PGM546_DRIFT 546.00 BOOL  ; PAST23 TIL T2009
PGM546_DRIFT_N5 2831.09 BOOL
PGM546_FEIL 546.04 BOOL  ; PAST23 TIL T2009
PGM546_FEILTID 546.05 BOOL  ; PAST23 TIL T2009
PGM546_FEILTID_S T0546 BOOL
PGM546_FEILTID_T 0546 NUMBER
PGM546_IKKE_FEIL_N5 2831.13 BOOL
PGM546_START 546.07 BOOL  ; PAST23 TIL T2009
PGM546_STOPP 546.09 BOOL  ; PAST23 TIL T2009
PGM546_STOPP_N5 2831.08 BOOL
PGM546_T2009_DREN_IND 1246.01 BOOL  ; DREN FRA V2347
PGM546_T2009_IND 1246.00 BOOL
PGM548_0_STATUS 548.01 BOOL  ; LAGER TIL T2030-DIREKTE-CONTAINER
PGM548_1_STATUS 548.02 BOOL  ; LAGER TIL T2030-DIREKTE-CONTAINER
PGM548_2030_IND 1248.00 BOOL
PGM548_2_STATUS 548.03 BOOL  ; LAGER TIL T2030-DIREKTE-CONTAINER
PGM548_CONT_IND 1248.02 BOOL
PGM548_DRIFT 548.00 BOOL  ; LAGER TIL T2030-DIREKTE-CONTAINER
PGM548_FEIL 548.04 BOOL  ; LAGER TIL T2030-DIREKTE-CONTAINER
PGM548_FEILTID 548.05 BOOL  ; LAGER TIL T2030-DIREKTE-CONTAINER
PGM548_INDIVID_INNE 548.15 BOOL  ; LAGER TIL T2030-DIREKTE-CONTAINER
PGM548_INDKON 548.06 BOOL  ; LAGER TIL T2030-DIREKTE-CONTAINER
PGM548_MODN_IND 1248.01 BOOL
PGM548_OFF_IMP 548.14 BOOL  ; LAGER TIL T2030-DIREKTE-CONTAINER
PGM548_ONIMPULS 548.11 BOOL  ; LAGER TIL T2030-DIREKTE-CONTAINER
PGM548_START 548.07 BOOL  ; LAGER TIL T2030-DIREKTE-CONTAINER
PGM548_STARTIMPULS 548.10 BOOL  ; LAGER TIL T2030-DIREKTE-CONTAINER
PGM548_STOPP 548.09 BOOL  ; LAGER TIL T2030-DIREKTE-CONTAINER
PGM548_TID_S T0548 BOOL  ; X
PGM548_TID_T 0548 NUMBER  ; X
PGM548_TMU_USIKRET 548.08 BOOL  ; LAGER TIL T2030-DIREKTE-CONTAINER
PGM550_START 550.07 BOOL  ; TGR10 TIL UHT
PGM5523_2_STATUS_N5 2810.11 BOOL
PGM552_0_STATUS 552.01 BOOL  ; PAST21 TIL T.GR08 OG T20.28-29
PGM552_1_STATUS 552.02 BOOL  ; PAST21 TIL T.GR08 OG T20.28-29
PGM552_1_STATUS_N5 2807.10 BOOL  ; PAST21 TIL T.GR08 OG T20.28-29
PGM552_2_STATUS 552.03 BOOL  ; PAST21 TIL T.GR08 OG T20.28-29
PGM552_2_STATUS_N5 2807.11 BOOL  ; PAST21 TIL T.GR08 OG T20.28-29
PGM552_DRIFT 552.00 BOOL  ; PAST21 TIL T.GR08 OG T20.28-29
PGM552_DRIFT_N5 2810.08 BOOL
PGM552_FEIL 552.04 BOOL  ; PAST21 TIL T.GR08 OG T20.28-29
PGM552_FEILTID 552.05 BOOL  ; PAST21 TIL T.GR08 OG T20.28-29
PGM552_FEILTID_T 0552 NUMBER
PGM552_IKKE_FEIL_N5 2810.12 BOOL  ; PAST21 TIL T.GR08 OG T20.28-29
PGM552_INDIVID_INNE 552.15 BOOL  ; PAST21 TIL T.GR08 OG T20.28-29
PGM552_INDKON 552.06 BOOL  ; PAST21 TIL T.GR08 OG T20.28-29
PGM552_IND_P21_T0801 1252.00 BOOL  ; TIL
PGM552_IND_P21_T0802 1252.01 BOOL
PGM552_IND_P21_T0803 1252.02 BOOL
PGM552_IND_P21_T0804 1252.03 BOOL
PGM552_IND_P21_T0805 1252.04 BOOL
PGM552_IND_P21_T2028 1252.05 BOOL
PGM552_IND_P21_T2029 1252.06 BOOL
PGM552_OFF_IMP 552.14 BOOL  ; PAST21 TIL T.GR08 OG T20.28-29
PGM552_ONIMPULS 552.11 BOOL  ; PAST21 TIL T.GR08 OG T20.28-29
PGM552_START 552.07 BOOL  ; PAST21 TIL T.GR08 OG T20.28-29
PGM552_STARTIMPULS 552.10 BOOL  ; PAST21 TIL T.GR08 OG T20.28-29
PGM552_STOPP 552.09 BOOL  ; PAST21 TIL T.GR08 OG T20.28-29
PGM552_STOPP_N5 2810.07 BOOL
PGM552_STOPP_S T0652 BOOL
PGM552_STOPP_T 0652 NUMBER
PGM552_TID_S T0552 BOOL  ; X
PGM552_TMU_USIKRET 552.08 BOOL  ; PAST21 TIL T.GR08 OG T20.28-29
PGM553_0_STATUS 553.01 BOOL  ; PAST21 TIL T.GR09
PGM553_0_STATUS_N5 2813.09 BOOL
PGM553_1_STATUS 553.02 BOOL  ; PAST21 TIL T.GR09
PGM553_1_STATUS_N5 2813.10 BOOL
PGM553_2_STATUS 553.03 BOOL  ; PAST21 TIL T.GR09
PGM553_2_STATUS_N5 2813.11 BOOL
PGM553_DRIFT 553.00 BOOL  ; PAST21 TIL T.GR09
PGM553_DRIFT_N5 2813.08 BOOL
PGM553_FEIL 553.04 BOOL  ; PAST21 TIL T.GR09
PGM553_FEILTID 553.05 BOOL  ; PAST21 TIL T.GR09
PGM553_FEILTID_T 0553 NUMBER
PGM553_IKKE_FEIL_N5 2813.12 BOOL
PGM553_IND_P21_T0901 1253.00 BOOL
PGM553_IND_P21_T0902 1253.01 BOOL
PGM553_IND_P21_T0903 1253.02 BOOL
PGM553_IND_P21_T0904 1253.03 BOOL
PGM553_IND_P21_T0905 1253.04 BOOL
PGM553_START 553.07 BOOL  ; PAST21 TIL T.GR09
PGM553_STOPP 553.09 BOOL  ; PAST21 TIL T.GR09
PGM553_STOPP_N5 2813.07 BOOL
PGM553_STOPP_S T0653 BOOL
PGM553_STOPP_T 0653 NUMBER
PGM553_TID_S T0553 BOOL  ; X
PGM553_TIL_TGR08_IND_N5 2808.00 BOOL
PGM553_TMU 553.08 BOOL  ; PAST21 TIL T.GR09
PGM5544_STARTIMPULS 544.10 BOOL  ; BIL TI OEKOMELKTANK T27.01
PGM554_0_STATUS 554.01 BOOL  ; PAST22 TIL T.GR08
PGM554_0_STATUS_N5 2813.02 BOOL
PGM554_1_STATUS 554.02 BOOL  ; PAST22 TIL T.GR08
PGM554_1_STATUS_N5 2813.03 BOOL
PGM554_2_STAT 554.03 BOOL  ; PAST22 TIL T.GR08
PGM554_2_STATUS_N5 2813.04 BOOL
PGM554_DRIFT 554.00 BOOL  ; PAST22 TIL T.GR08
PGM554_DRIFT_N5 2813.01 BOOL
PGM554_FEIL 554.04 BOOL  ; PAST22 TIL T.GR08
PGM554_FEILTID 554.05 BOOL  ; PAST22 TIL T.GR08
PGM554_FEILTID_T 0554 NUMBER
PGM554_IKKE_FEIL_N5 2813.05 BOOL
PGM554_IND_P22_T0801 1254.00 BOOL  ; TIL
PGM554_IND_P22_T0802 1254.01 BOOL
PGM554_IND_P22_T0803 1254.02 BOOL
PGM554_IND_P22_T0804 1254.03 BOOL
PGM554_IND_P22_T0805 1254.04 BOOL
PGM554_IND_P22_T2028 1254.05 BOOL
PGM554_IND_P22_T2029 1254.06 BOOL
PGM554_START 554.07 BOOL  ; PAST22 TIL T.GR08
PGM554_STOPP 554.09 BOOL  ; PAST22 TIL T.GR08
PGM554_STOPP_N5 2813.00 BOOL
PGM554_STOPP_S T0654 BOOL
PGM554_STOPP_T 0654 NUMBER
PGM554_TID_S T0554 BOOL  ; X
PGM555_0_STATUS 555.01 BOOL  ; PAST22 TIL T.GR09
PGM555_0_STATUS_N5 2814.02 BOOL
PGM555_1_STATUS 555.02 BOOL  ; PAST22 TIL T.GR09
PGM555_1_STATUS_N5 2814.03 BOOL
PGM555_2_STATUS 555.03 BOOL  ; PAST22 TIL T.GR09
PGM555_2_STATUS_N5 2814.04 BOOL
PGM555_DRIFT 555.00 BOOL  ; PAST22 TIL T.GR09
PGM555_DRIFT_N5 2814.01 BOOL
PGM555_FEIL 555.04 BOOL  ; PAST22 TIL T.GR09
PGM555_FEILTID 555.05 BOOL  ; PAST22 TIL T.GR09
PGM555_FEILTID_T 0555 NUMBER
PGM555_IKKE_FEIL_N5 2814.05 BOOL
PGM555_IND_P22_T0901 1255.00 BOOL  ; '
PGM555_IND_P22_T0902 1255.01 BOOL
PGM555_IND_P22_T0903 1255.02 BOOL
PGM555_IND_P22_T0904 1255.03 BOOL
PGM555_IND_P22_T0905 1255.04 BOOL
PGM555_IND_P22_TGR11 1255.05 BOOL
PGM555_START 555.07 BOOL  ; PAST22 TIL T.GR09
PGM555_STOPP 555.09 BOOL  ; PAST22 TIL T.GR09
PGM555_STOPP_N5 2814.00 BOOL
PGM555_STOPP_S T0655 BOOL  ; X
PGM555_STOPP_T 0555 NUMBER
PGM555_TID_S T0555 BOOL  ; X
PGM556_0_STATUS 556.01 BOOL  ; PAST23 TIL T.GR10
PGM556_0_STATUS_N5 2814.09 BOOL
PGM556_1_STATUS 556.02 BOOL  ; PAST23 TIL T.GR10
PGM556_1_STATUS_N5 2814.10 BOOL
PGM556_2_STATUS 556.03 BOOL  ; PAST23 TIL T.GR10
PGM556_2_STATUS_N5 2814.11 BOOL
PGM556_DRENSTID_S T0688 BOOL
PGM556_DRENSTID_T 0688 NUMBER
PGM556_DRIFT 556.00 BOOL  ; PAST23 TIL T.GR10
PGM556_DRIFT_N5 2814.08 BOOL
PGM556_FEIL 556.04 BOOL  ; PAST23 TIL T.GR10
PGM556_FEILTID 556.05 BOOL  ; PAST23 TIL T.GR10
PGM556_FEILTID_T 0556 NUMBER
PGM556_IKKE_FEIL_N5 2814.12 BOOL
PGM556_IND_DREN 1256.04 BOOL
PGM556_IND_P23_DREN 1256.03 BOOL
PGM556_IND_P23_T1002 1256.00 BOOL
PGM556_IND_P23_T1003 1256.01 BOOL
PGM556_IND_P23_T1004 1256.02 BOOL
PGM556_START 556.07 BOOL  ; PAST23 TIL T.GR10
PGM556_STOPP 556.09 BOOL  ; PAST23 TIL T.GR10
PGM556_STOPP_N5 2814.07 BOOL
PGM556_STOPP_S T0656 BOOL
PGM556_STOPP_T 0656 NUMBER
PGM556_TID_S T0556 BOOL  ; X
PGM556_TMU 556.08 BOOL  ; PAST23 TIL T.GR10
PGM557_0_STATUS 557.01 BOOL  ; V3345 TIL T2033-34-35-DIREKTE
PGM557_1_STATUS 557.02 BOOL  ; V3345 TIL T2033-34-35-DIREKTE
PGM557_2_STAT 557.03 BOOL  ; V3345 TIL T2033-34-35-DIREKTE
PGM557_DIREKTE_VALG 357.03 BOOL  ; INDIVIDVALG FRA KOEREGISTER.
PGM557_DRIFT 557.00 BOOL  ; V3345 TIL T2033-34-35-DIREKTE
PGM557_FEIL 557.04 BOOL  ; V3345 TIL T2033-34-35-DIREKTE
PGM557_FEILTID 557.05 BOOL  ; V3345 TIL T2033-34-35-DIREKTE
PGM557_INDIVID_INNE 557.15 BOOL  ; V3345 TIL T2033-34-35-DIREKTE
PGM557_INDKON 557.06 BOOL  ; V3345 TIL T2033-34-35-DIREKTE
PGM557_KOELES 357.14 BOOL  ; SPERR INNLESNING TIL KOE-REGISTER.
PGM557_KOMMANDO_KOE 357.15 BOOL  ; D3000 VERDI KAN OVERFOERES TIL KOE-REGISTER.
PGM557_OFF_IMP 557.14 BOOL  ; V3345 TIL T2033-34-35-DIREKTE
PGM557_ONIMPULS 557.11 BOOL  ; V3345 TIL T2033-34-35-DIREKTE
PGM557_START 557.07 BOOL  ; V3345 TIL T2033-34-35-DIREKTE
PGM557_STARTIMPULS 557.10 BOOL  ; V3345  TIL T2033-34-35-DIREKTE
PGM557_STOPP 557.09 BOOL  ; V3345 TIL T2033-34-35-DIREKTE
PGM557_T2033_VALG 357.00 BOOL  ; INDIVIDVALG FRA KOEREGISTER.
PGM557_T2034_VALG 357.01 BOOL  ; INDIVIDVALG FRA KOEREGISTER.
PGM557_T2035_VALG 357.02 BOOL  ; INDIVIDVALG FRA KOEREGISTER.
PGM557_TID_S T0557 BOOL  ; X
PGM557_TID_T 0557 NUMBER  ; X
PGM557_TIL_DIREKTE_IND 1257.03 BOOL
PGM557_TIL_T2033_IND 1257.00 BOOL
PGM557_TIL_T2034_IND 1257.01 BOOL  ; X
PGM557_TIL_T2035_IND 1257.02 BOOL
PGM557_TMU_USIKRET 557.08 BOOL  ; V3345 TIL T2033-34-35-DIREKTE
PGM558_0_STATUS 558.01 BOOL  ; V3335 TIL T2033-34-35-DIREKTE
PGM558_1_STATUS 558.02 BOOL  ; V3335 TIL T2033-34-35-DIREKTE
PGM558_2_STAT 558.03 BOOL  ; V3335 TIL T2033-34-35-DIREKTE
PGM558_DIREKTE_VALG 358.03 BOOL  ; INDIVIDVALG FRA KOEREGISTER.
PGM558_FEIL 558.04 BOOL  ; V3335 TIL T2033-34-35-DIREKTE
PGM558_FEILTID 558.05 BOOL  ; V3335 TIL T2033-34-35-DIREKTE
PGM558_INDIVID_INNE 558.15 BOOL  ; V3385 TIL T2033-34-35-DIREKTE
PGM558_INDKON 558.06 BOOL  ; V3335 TIL T2033-34-35-DIREKTE
PGM558_KOELES 358.14 BOOL  ; SPERR INNLESNING TIL KOE-REGISTER.
PGM558_KOMMANDO_KOE 358.15 BOOL  ; D3000 VERDI KAN OVERFOERES TIL KOE-REGISTER.
PGM558_OFF_IMP 558.14 BOOL  ; V3335 TIL T2033-34-35-DIREKTE
PGM558_ONIMPULS 558.11 BOOL  ; V3335 TIL T2033-34-35-DIREKTE
PGM558_START 558.07 BOOL  ; V3335 TIL T2033-34-35-DIREKTE
PGM558_STARTIMPULS 558.10 BOOL  ; V3335  TIL T2033-34-35-DIREKTE
PGM558_STOPP 558.09 BOOL  ; V3335 TIL T2033-34-35-DIREKTE
PGM558_T2033_VALG 358.00 BOOL  ; INDIVIDVALG FRA KOEREGISTER.
PGM558_T2034_VALG 358.01 BOOL  ; INDIVIDVALG FRA KOEREGISTER.
PGM558_T2035_VALG 358.02 BOOL  ; INDIVIDVALG FRA KOEREGISTER.
PGM558_TID_S T0558 BOOL  ; X
PGM558_TID_T 0558 NUMBER  ; X
PGM558_TIL_DIREKTE_IND 1258.03 BOOL
PGM558_TIL_T2033_IND 1258.00 BOOL
PGM558_TIL_T2034_IND 1258.01 BOOL  ; X
PGM558_TIL_T2035_IND 1258.02 BOOL
PGM558_TMU_USIKRET 558.08 BOOL  ; V3335 TIL T2033-34-35-DIREKTE
PGM559_0_STATUS 559.01 BOOL
PGM559_0_STATUS_N5 2822.02 BOOL
PGM559_1_STATUS 559.02 BOOL
PGM559_1_STATUS_N5 2822.03 BOOL
PGM559_2_STATUS 559.03 BOOL
PGM559_2_STATUS_N5 2822.04 BOOL
PGM559_DRIFT 559.00 BOOL
PGM559_DRIFT_N5 2822.01 BOOL
PGM559_FEIL 559.04 BOOL
PGM559_FEILTID 559.05 BOOL
PGM559_IKKE_FEIL_N5 2822.05 BOOL
PGM559_P21_TIL_RETURT_IND 1259.00 BOOL
PGM559_START 559.07 BOOL
PGM559_STOPP 559.09 BOOL
PGM559_STOPP_S T0659 BOOL
PGM559_STOPP_T 0659 NUMBER
PGM559_STOP_N5 2822.00 BOOL
PGM559_TID_S T0559 BOOL  ; X
PGM559_TMU 559.08 BOOL
PGM560_0_STATUS 560.01 BOOL
PGM560_0_STATUS_N5 2822.09 BOOL
PGM560_1_STATUS 560.02 BOOL
PGM560_1_STATUS_N5 2822.10 BOOL
PGM560_2_STATUS 560.03 BOOL
PGM560_2_STATUS_N5 2822.11 BOOL
PGM560_DRIFT 560.00 BOOL
PGM560_DRIFT_N5 2822.08 BOOL
PGM560_FEIL 560.04 BOOL
PGM560_FEILTID 560.05 BOOL
PGM560_IKKE_FEIL_N5 2822.12 BOOL
PGM560_P22_TIL_RETURT_IND 1260.00 BOOL
PGM560_START 560.07 BOOL
PGM560_STOPP 560.09 BOOL
PGM560_STOPP_N5 2822.07 BOOL
PGM560_STOPP_S T0760 BOOL
PGM560_STOPP_T 0760 NUMBER
PGM560_TID_S T0560 BOOL  ; X
PGM560_TID_T 0560 NUMBER
PGM560_TMU 560.08 BOOL
PGM561_0_STATUS 561.01 BOOL
PGM561_0_STATUS_N5 2818.11 BOOL
PGM561_1_STATUS 561.02 BOOL
PGM561_1_STATUS_N5 2818.12 BOOL
PGM561_2_STATUS 561.03 BOOL
PGM561_2_STATUS_N5 2818.13 BOOL
PGM561_DRIFT 561.00 BOOL
PGM561_DRIFT_N5 2818.10 BOOL
PGM561_FEIL 561.04 BOOL
PGM561_FEILTID 561.05 BOOL
PGM561_IKKE_FEIL_N5 2818.14 BOOL
PGM561_P21_TIL_T2009_IND 1261.00 BOOL
PGM561_START 561.07 BOOL
PGM561_STOPP 561.09 BOOL
PGM561_STOPP_N5 2818.09 BOOL
PGM561_STOPP_S T0761 BOOL
PGM561_STOPP_T 0761 NUMBER
PGM561_TID_S T0561 BOOL
PGM561_TID_T 561 LWORD
PGM561_TMU 561.08 BOOL
PGM562_0_STATUS 562.01 BOOL  ; T20.09>P23
PGM562_0_STATUS_N5 2819.11 BOOL
PGM562_1_STATUS 562.02 BOOL  ; T20.09>P23
PGM562_1_STATUS_N5 2819.12 BOOL
PGM562_2_STAT 562.03 BOOL  ; T20.09>P23
PGM562_2_STAT_N5 2819.13 BOOL
PGM562_DRIFT 562.00 BOOL  ; T20.09>P23
PGM562_DRIFT_N5 2819.10 BOOL
PGM562_FEIL 562.04 BOOL  ; T20.09>P23
PGM562_FEILTID 562.05 BOOL  ; T20.09>P23
PGM562_IKKE_FEIL_N5 2819.14 BOOL  ; 1= IKKE FEIL
PGM562_INDKON 562.06 BOOL  ; T20.09>P23
PGM562_IND_T2009 1262.00 BOOL  ; T20.09>P23
PGM562_RESET_N5 2819.09 BOOL
PGM562_START 562.07 BOOL  ; T20.09>P23
PGM562_STOPP 562.09 BOOL  ; T20.09>P23
PGM562_STOPP_S T0826 BOOL
PGM562_STOPP_T 0826 NUMBER
PGM562_TID_S T0562 BOOL
PGM562_TID_T 0562 NUMBER
PGM562_TMU 562.08 BOOL  ; T20.09>P23
PGM584_0_STATUS 584.01 BOOL  ; XX
PGM584_1_STATUS 584.02 BOOL  ; Z
PGM584_2_STATUS 584.03 BOOL  ; Z
PGM584_DRIFT 584.00 BOOL  ; XX
PGM584_FEIL 584.04 BOOL  ; Z
PGM584_FEILTID 584.05 BOOL  ; Z
PGM584_FEILTID_S T0584 BOOL
PGM584_FEILTID_T 0584 NUMBER
PGM584_INDKON 584.06 BOOL  ; Z
PGM584_IND_INNE 584.15 BOOL  ; Z
PGM584_IND_T40 1284.00 BOOL  ; Z
PGM584_IND_T40_VALG 384.00 BOOL  ; Z
PGM584_IND_T41 1284.01 BOOL  ; Z
PGM584_IND_T41_VALG 384.01 BOOL  ; Z
PGM584_KOELES 384.14 BOOL  ; Z
PGM584_KOEPLASS_1 D5256 CHANNEL  ; XFOERST I KOE
PGM584_KOEPLASS_2 D5257 CHANNEL
PGM584_KOEPLASS_3 D5258 CHANNEL  ; X
PGM584_KOMMANDO_KOE 384.15 BOOL  ; Z
PGM584_OFF_IMPULS 584.14 BOOL  ; Z
PGM584_ONIMPULS 584.11 BOOL  ; Z
PGM584_RESET 584.09 BOOL  ; Z
PGM584_START 584.07 BOOL  ; Z
PGM584_STARTIMPULS 584.10 BOOL  ; Z
PGM584_TMU 584.08 BOOL
PGM584_TMU_TID_S T0784 BOOL  ; MAX-TID TMU OM IKKE LINJE LEGGES
PGM584_TMU_TID_T 0784 NUMBER  ; MAX-TID TMU OM IKKE LINJE LEGGES
PGM585_0_STATUS 585.01 BOOL  ; XX
PGM585_1_STATUS 585.02 BOOL  ; Z
PGM585_2_STATUS 585.03 BOOL  ; Z
PGM585_DRIFT 585.00 BOOL
PGM585_FEIL 585.04 BOOL  ; Z
PGM585_FEILTID 585.05 BOOL  ; Z
PGM585_FEILTID_S T0585 BOOL
PGM585_FEILTID_T 0585 NUMBER
PGM585_INDKON 585.06 BOOL  ; Z
PGM585_IND_INNE 585.15 BOOL  ; Z
PGM585_IND_T40 1285.00 BOOL  ; Z
PGM585_IND_T40_VALG 385.00 BOOL  ; Z
PGM585_IND_T41 1285.01 BOOL  ; Z
PGM585_IND_T41_VALG 385.01 BOOL  ; Z
PGM585_KOELES 385.14 BOOL  ; Z
PGM585_KOEPLASS_1 D5260 CHANNEL  ; XFOERST I KOE
PGM585_KOEPLASS_2 D5261 CHANNEL
PGM585_KOEPLASS_3 D5262 CHANNEL  ; X
PGM585_KOMMANDO_KOE 385.15 BOOL  ; Z
PGM585_OFF_IMPULS 585.14 BOOL  ; Z
PGM585_ONIMPULS 585.11 BOOL  ; Z
PGM585_RESET 585.09 BOOL  ; Z
PGM585_START 585.07 BOOL  ; Z
PGM585_STARTIMPULS 585.10 BOOL  ; Z
PGM585_TMU 585.08 BOOL
PGM585_TMU_TID_S T0785 BOOL  ; MAX-TID TMU OM IKKE LINJE LEGGES
PGM585_TMU_TID_T 0785 NUMBER  ; MAX-TID TMU OM IKKE LINJE LEGGES
PGM585_TOEM_BIL 585.13 BOOL  ; START TOEMMING FRA MOTTAK
PGM586_0_STATUS 586.01 BOOL  ; XX
PGM586_1_STATUS 586.02 BOOL  ; Z
PGM586_2_STATUS 586.03 BOOL  ; Z
PGM586_DRIFT 586.00 BOOL
PGM586_FEIL 586.04 BOOL  ; Z
PGM586_FEILTID 586.05 BOOL  ; Z
PGM586_FEILTID_S T0586 BOOL
PGM586_FEILTID_T 0586 NUMBER
PGM586_INDKON 586.06 BOOL  ; Z
PGM586_IND_INNE 586.15 BOOL  ; Z
PGM586_IND_PAST21 1286.00 BOOL
PGM586_IND_PAST21_VALG 386.00 BOOL  ; Z
PGM586_IND_PAST22 1286.01 BOOL
PGM586_IND_PAST22_VALG 386.01 BOOL  ; Z
PGM586_KOELES 386.14 BOOL  ; Z
PGM586_KOMMANDO_KOE 386.15 BOOL  ; Z
PGM586_OFF_IMPULS 586.14 BOOL  ; Z
PGM586_ONIMPULS 586.11 BOOL
PGM586_RES 586.13 BOOL
PGM586_RESET 586.09 BOOL  ; Z
PGM586_START 586.07 BOOL  ; Z
PGM586_STARTIMPULS 586.10 BOOL
PGM586_TMU 586.08 BOOL
PGM586_TMU_TID_S T0786 BOOL  ; MAX-TID TMU OM IKKE LINJE LEGGES
PGM586_TMU_TID_T 0786 NUMBER  ; MAX-TID TMU OM IKKE LINJE LEGGES
PGM_515_3040_N6 2802.13 BOOL
PLS_FORSINKET_START_T T0905 BOOL  ; FORSINKET STARTSIGNAL 999.06  VED OPPSTART AV PLS
PLS_INNFORSINK 999.06 BOOL  ; FORSINKET SIGNAL VED OPPSTART AV pls
PORT_0 A202.00 BOOL
PORT_2 A202.02 BOOL
PRESET_REG_1 D20000 CHANNEL
PRESET_REG_2 D20050 CHANNEL
PRESET_REG_3 D20100 CHANNEL
PRESET_REG_5 D20200 CHANNEL
PRESET_REG_6 D20250 CHANNEL
PT INT
P_8001_MANUELL 1000.00 BOOL
P_8002_MANUELL 1000.01 BOOL
P_8003_MANUELL 1000.02 BOOL
Q0101_DRIFT 2228.00 BOOL  ; Z
Q0101_FLOW_INN D1692 REAL  ; Z
Q0101_HJ D2050 INT
Q0101_MENGDE_INN D1690 REAL  ; Z
Q0101_RESET 2228.01 BOOL  ; Z
Q0101_RESET_S T0063 BOOL
Q0101_RESET_T 0063 NUMBER
Q0111_DRIFT 2228.02 BOOL  ; Z
Q0111_FLOW_INN D1698 REAL  ; Z
Q0111_MENGDE_INN D1696 REAL  ; Z
Q0111_RESET 2228.03 BOOL  ; Z
Q0111_RESET_S T0064 BOOL
Q0111_RESET_T 0064 NUMBER
Q0201_DRIFT 2228.04 BOOL  ; Z
Q0201_FLOW_INN D1704 REAL  ; Z
Q0201_HJ D2054 REAL
Q0201_MENGDE_INN D1702 REAL  ; Z
Q0201_RESET 2228.05 BOOL  ; Z
Q0211_DRIFT 2228.06 BOOL  ; Z
Q0211_FLOW_INN D1710 REAL  ; Z
Q0211_MENGDE_INN D1708 REAL  ; Z
Q0211_RESET 2228.07 BOOL  ; Z
Q06_FLOW_OMR D6070 REAL  ; B0605
Q06_FLOW_RAA D6072 REAL  ; B0605
Q201_RESET_S T0065 BOOL
Q201_RESET_T 0065 NUMBER
Q2022_DRIFT_PR2 5012.00 BOOL  ; MENGDE VED OVERKJOERING FRA T20.02-05 DIREKTE TIL T20.11-19   DRIFTSIGNAL
Q2022_OPN_FORV 694.15 BOOL
Q2022_ORD1_AV_4_PR2 5120 UINT  ; PT L2-2
Q2022_ORD2_AV_4_PR2 5121 UINT  ; PT ISVANN L1
Q2022_ORD3_AV_4_PR2 5122 UINT  ; PT ISVANN L2
Q2022_ORD4_AV_4_PR2 5123 UINT  ; MENGDE VED OVERKJOERING FRA T20.02-05 DIREKTE TIL T20.11-19
Q2022_RESET_PR2 5012.08 BOOL  ; MENGDE VED OVERKJOERING FRA T20.02-05 DIREKTE TIL T20.11-19   RESETSIGNAL
Q211_RESET_S T0066 BOOL
Q211_RESET_T 0066 NUMBER
Q21_DRIFT 2227.06 BOOL  ; Z
Q21_FORV_OK 4803.14 BOOL  ; Q21 FORVALG OPNAADD
Q21_MENGDE_TGR08 D3608 DINT  ; KJOERT MENGDE TIL TGR08
Q21_MENGDE_TGR09 D3610 DINT  ; KJOERT MENGDE TIL TGR09
Q21_MENGDE_UHT D3612 DINT  ; KJOERT MENGDE TIL UHT
Q21_RESET 2227.07 BOOL  ; Z
Q21_RESET_FORV 4803.15 BOOL  ; RESET TELLER VED OPNAADD FORVALG
Q21_SIST_KJ_MENGDE D3616 DINT  ; SIST KJOERTE MENGDE
Q21__LITERIMP 2527.06 BOOL  ; Z
Q22_DRIFT 2227.08 BOOL
Q22_FORV_OK 4813.14 BOOL  ; Q22 FORVALG OPNAADD
Q22_MENGDE_TGR08 D3708 DINT  ; KJOERT MENGDE TIL TGR08
Q22_MENGDE_TGR09 D3710 DINT  ; KJOERT MENGDE TIL TGR09
Q22_MENGDE_UHT D3712 DINT  ; KJOERT MENGDE TIL UHT
Q22_RESET 2227.09 BOOL
Q22_RESET_FORV 4813.15 BOOL  ; RESET TELLER VED OPNAADD FORVALG
Q22_SIST_KJ_MENGDE D3716 DINT  ; SIST KJOERTE MENGDE
Q22__LITERIMP 2527.08 BOOL  ; Z
Q23_DRIFT 2227.10 BOOL
Q23_FORV_OK 4823.14 BOOL  ; Q23 FORVALG OPNAADD
Q23_MENGDE_T1002 D3808 DINT  ; KJOERT MENGDE TIL T10.02
Q23_MENGDE_T1003 D3810 DINT  ; KJOERT MENGDE TIL T10.03
Q23_MENGDE_T1004 D3812 DINT  ; KJOERT MENGDE TIL T10.04
Q23_RESET 2227.11 BOOL
Q23_RESET_FORV 4823.15 BOOL  ; RESET TELLER VED OPNAADD FORVALG
Q23_RESET_S T0824 BOOL
Q23_RESET_T 0824 NUMBER
Q23_SIST_KJ_MENGDE D3816 DINT  ; SIST KJOERTE MENGDE
Q23__LITERIMP 2527.10 BOOL  ; Z
Q8001_DRIFT 2227.00 BOOL  ; DRIFTSIGNAL TIL MAALER
Q8001_ER_FLOW_M3 D8050 INT
Q8001_ER_FLOW_M3FLYT D8822 REAL
Q8001_ER_M3 D8050 INT
Q8001_FLOW_INN D1640 REAL
Q8001_MENGDE_INN D1650 REAL  ; 0,1xRIKTIG MENGDE
Q8001_RESET 2227.01 BOOL  ; RESETSIGNAL TIL MAALER
Q8001_RESETTID T0150 BOOL  ; TID SOM RESETSIGN. LIGGER INNE
Q8002_DRIFT 2227.02 BOOL
Q8002_ER_FLOW_M3 D8052 INT
Q8002_ER_FLOW_M3FLYT D8824 REAL
Q8002_FLOW_INN D1642 REAL
Q8002_MENGDE_INN D1652 REAL  ; 0,1xRIKTIG MENGDE
Q8002_RESET 2227.03 BOOL
Q8002_RESETTID T0250 BOOL  ; TID SOM RESETSIGN. LIGGER INNE
Q8003_DRIFT 2227.04 BOOL
Q8003_ER_FLOW_M3 D8054 INT
Q8003_ER_FLOW_M3FLYT D8826 REAL
Q8003_FLOW_INN D1644 REAL
Q8003_MENGDE_INN D1654 REAL  ; 0,1xRIKTIG MENGDE
Q8003_RESET 2227.05 BOOL
Q8003_RESETTID T0350 BOOL  ; TID SOM RESETSIGN. LIGGER INNE
Q8014_MENGDE_DRIFT 2208.06 BOOL  ; DRIFTSIGNAL TIL MAALER
Q8014_MENGDE_RESET 2208.07 BOOL  ; RESETSIGNAL TIL MAALER
Q8017_RESETTID T0154 BOOL  ; TID SOM RESETSIGN. LIGGER INNE
R2801_UT_N6 2864.02 BOOL
R2901_UT_N6 2864.03 BOOL
REGN1_P8001 D20044 REAL
REGN1_P8002 D20144 REAL
REGN1_P8003 D20244 REAL
REGN1_V8014 D20094 REAL
REGN1_V8024 D20194 REAL
REGN1_V8034 D20294 REAL
REGN2_P8001 D20046 REAL
REGN2_P8002 D20146 REAL
REGN2_P8003 D20246 REAL
REGN2_V8014 D20096 REAL
REGN2_V8024 D20196 REAL
REGN2_V8034 D20296 REAL
REGN_ANALOG_K1 D8902 REAL
REGN_ANALOG_K2 D8904 REAL
REGN_ANALOG_K3 D8906 REAL
REGN_HJ_REGISTER D8900 UINT
REG_P2104_SISTE_KONTR_ORD D22388 CHANNEL
REG_V2161_SISTE_KONTR_ORD D22088 CHANNEL
REG_V2353 BRA_PID_INV
RET_STENGT_VST90_K3_N5 2859.05 BOOL
RV0301_AUTO 1054.15 BOOL
RV0301_DR_TID_C C0060 BOOL
RV0301_DR_TID_S C60 CHANNEL
RV0301_INN 2701.01 BOOL  ; Z
RV0301_MAN 1004.15 BOOL
RV0301_STOPP_TID_C C0061 BOOL
RV0301_STOPP_TID_S C61 CHANNEL
RV0301_UT 2401.01 BOOL  ; Z
RV0301__VALGT 601.05 BOOL
RV0401_AUTO 1055.05 BOOL  ; LITE RV
RV0401_DREN_TID_AUTO C0078 BOOL  ; LITE RV
RV0401_DR_TID_C C0066 BOOL  ; LITE RV
RV0401_DR_TID_S C66 CHANNEL  ; LITE RV
RV0401_INN 2702.05 BOOL  ; LITE RV
RV0401_MAN 1005.05 BOOL  ; LITE RV
RV0401_STOPP_TID_AUTO C0079 BOOL  ; LITE RV
RV0401_STOPP_TID_C C0067 BOOL  ; LITE RV
RV0401_STOPP_TID_S C67 CHANNEL  ; LITE RV
RV0401_UT 2402.05 BOOL  ; LITE RV
RV0401_VALGT 603.05 BOOL  ; LITE RV
RV0401__VALGT 603.05 BOOL  ; LITE RV
RV0402_AUTO 1055.06 BOOL  ; STORT RV
RV0402_DREN_TID_AUTO C0080 BOOL  ; STORT RV
RV0402_DR_TID_C C0076 BOOL  ; STORT RV
RV0402_DR_TID_S C76 CHANNEL  ; STORT RV
RV0402_INN 2702.06 BOOL  ; STORT RV
RV0402_MAN 1005.06 BOOL  ; STORT RV
RV0402_STOPP_TID_AUTO C0081 BOOL  ; STORT RV
RV0402_STOPP_TID_C C0077 BOOL  ; STORT RV
RV0402_STOPP_TID_S C77 CHANNEL  ; STORT RV
RV0402_UT 2402.06 BOOL  ; STORT RV
RV0402_VALGT 603.10 BOOL  ; STORT RV
RV0402__VALGT 603.10 BOOL  ; STORT RV
RV0501_AUTO 1057.00 BOOL  ; LITE RV
RV0501_DREN_TID_AUTO C0082 BOOL  ; LITE RV
RV0501_DR_TID_C C0087 BOOL  ; LITE RV
RV0501_INN 2703.00 BOOL
RV0501_MAN 1007.00 BOOL  ; LITE RV
RV0501_STOPP_TID_AUTO C0083 BOOL  ; LITE RV
RV0501_STOPP_TID_C C0088 BOOL  ; LITE RV
RV0501_UT 2403.00 BOOL  ; LITE RV
RV0501_VALGT 606.00 BOOL  ; LITE RV
RV0502_AUTO 1057.01 BOOL  ; STORT RV
RV0502_DREN_TID_AUTO C0084 BOOL  ; STORT RV
RV0502_DR_TID_C C0089 BOOL  ; STORT RV
RV0502_INN 2703.01 BOOL
RV0502_MAN 1007.01 BOOL  ; STORT RV
RV0502_STOPP_TID_AUTO C0085 BOOL  ; STORT RV
RV0502_STOPP_TID_C C0090 BOOL  ; STORT RV
RV0502_UT 2403.01 BOOL  ; STORT RV
RV0502_VALGT 606.01 BOOL  ; STORT RV
RV2013_01_HOEY_INN_N5 2804.01 BOOL
RV2013_01_LAV_INN_N5 2804.00 BOOL
RV2013_02_INN_N5 2804.02 BOOL
RV2014_01_HOEY_INN_N5 2804.04 BOOL  ; HOEY HASTIGHET
RV2014_01_LAV_INN_N5 2804.03 BOOL
RV2014_02_INN_N5 2804.05 BOOL
RV2036_01_AUTO 1055.01 BOOL
RV2036_01_FUNKSJ H68.00 BOOL
RV2036_01_INN 2702.00 BOOL
RV2036_01_MAN 1005.01 BOOL
RV2036_01_UT 2402.00 BOOL
RV2036_ACC_HAST D6068 CHANNEL  ; 0-1000
RV2036_ACC_HAST_REG1 D18000 REAL
RV2036_ACC_HAST_REG2 D18002 REAL
RV2036_HAST D1458 ULINT_BCD  ; RAAVERDI
RV2036_PRS_HAST D6066 CHANNEL
RV2037_01_AUTO 1055.02 BOOL
RV2037_01_INN 2702.01 BOOL
RV2037_01_MAN 1005.02 BOOL
RV2037_01_UT 2402.01 BOOL
RV2037_ACC_HAST D6088 CHANNEL  ; 0-1000
RV2037_ACC_HAST_REG1 D18004 REAL
RV2037_ACC_HAST_REG2 D18006 REAL
RV2037_FUNKSJ H70.00 BOOL
RV2037_HAST D1460 WORD  ; RAAVERDI
RV2037_PRS_HAST D6086 CHANNEL
RV20_07_01_I_DR_N5 2820.13 BOOL  ; T20.07UHT AVD. INNG. DRIFT
RV20_11_01_I_DR_N5 2821.00 BOOL  ; T20.11UHT AVD. INNG. DRIFT
RV20_12_01_I_DR_N5 2821.01 BOOL  ; T20.12UHT AVD. INNG. DRIFT
RV20_33_01_I_DR_N5 2820.10 BOOL  ; T20.33 UHT AVD. INNG. DRIFT
RV20_34_01_I_DR_N5 2820.11 BOOL  ; T20.34 UHT AVD. INNG. DRIFT
RV20_35_01_DR_N5 2820.12 BOOL  ; T20.35UHT AVD. INNG. DRIFT
RV4001_AUTO 1055.12 BOOL
RV4001_INN 2702.07 BOOL
RV4001_MAN 1005.12 BOOL
RV4001_UT 2402.07 BOOL
RV4101_AUTO 1055.13 BOOL
RV4101_INN 2702.08 BOOL
RV4101_MAN 1005.13 BOOL
RV4101_UT 2402.08 BOOL
R_SWAP_HJELPEORD D122 CHANNEL
SCAN_1_KONTR_S T0055 BOOL
SCAN_1_KONTR_T 0055 NUMBER
SCAN_INN_KONTR_S T0842 BOOL  ; 1_SCAN_FORSINKER
SEND_0 993.00 BOOL
SEND_2 1994.01 BOOL
SEND_C0 D1100 CHANNEL
SEND_C1 D1101 CHANNEL
SEND_C2 D1102 CHANNEL
SEND_C3 D1103 CHANNEL
SEND_C4 D1104 CHANNEL
SEND_N6_C0 D1120 CHANNEL
SEND_N6_C1 D1121 CHANNEL
SEND_N6_C2 D1122 CHANNEL
SEND_N6_C3 D1123 CHANNEL
SEND_N6_C4 D1124 CHANNEL
SEP21_ALARM_CMD 4508.12 BOOL  ; Legge paa H-bit?
SEP21_ALARM_RESET 4508.13 BOOL  ; BYTTE DENNE I CIO 999
SEP21_ALARM_STOP 4506.09 BOOL
SEP21_ALARM_WDOG 4506.10 BOOL
SEP21_AUTO 1055.08 BOOL
SEP21_CIP_VANN 4505.00 BOOL
SEP21_CIP_VANN_OK 4506.04 BOOL
SEP21_CIP_VASKEM 4505.01 BOOL
SEP21_CIP_VASKEM_OK 4506.05 BOOL
SEP21_CMD_BUSY 4508.10 BOOL
SEP21_CMD_CIP_VANN_GITT 4508.03 BOOL
SEP21_CMD_CIP_VM_GITT 4508.04 BOOL
SEP21_CMD_FEED_OFF_GITT 4508.01 BOOL
SEP21_CMD_GITT 4508.09 BOOL
SEP21_CMD_PARTIALSK_GITT 4508.06 BOOL
SEP21_CMD_PRODUKT_1_GITT 4508.02 BOOL
SEP21_CMD_PRODUKT_2_GITT 4508.14 BOOL
SEP21_CMD_PROD_1_SLUTT_GITT 4508.08 BOOL
SEP21_CMD_PROD_2_SLUTT_GITT 4508.15 BOOL
SEP21_CMD_STANDBY_START_GITT 4508.00 BOOL
SEP21_CMD_START_MOT_GITT 4506.13 BOOL
SEP21_CMD_STOP_MOT_GITT 4508.07 BOOL
SEP21_CMD_TOTALSK_GITT 4508.05 BOOL
SEP21_DRIFT 4501.07 BOOL
SEP21_DRIFT_OK 4501.06 BOOL
SEP21_FEED_OFF_OK 4506.11 BOOL
SEP21_FEIL 4501.09 BOOL
SEP21_FEIL_KOM 3100.02 BOOL
SEP21_FRYSMODUS 4501.10 BOOL
SEP21_GLOBAL_STOP_REG_SEND_INN 4710 CHANNEL
SEP21_GL_ID_REG D116 INT
SEP21_GL_ID_REG_SEND D100 INT
SEP21_GL_ID_REG_SEND_INN 4701 INT
SEP21_GL_ID_REG_UT 4707 INT
SEP21_GL_START_REG D118 INT
SEP21_GL_START_REG_SEND D102 INT
SEP21_GL_START_REG_SEND_INN 4702 INT
SEP21_GL_START_REG_UT 4708 INT
SEP21_GL_STOP_REG D120 INT
SEP21_GL_STOP_REG_SEND D112 INT
SEP21_GL_STOP_REG_UT 4709 INT
SEP21_HANDSHAKE_OK 4508.11 BOOL
SEP21_INN 2700.15 BOOL
SEP21_I_LINJE 4500.06 BOOL
SEP21_MAN 1005.08 BOOL
SEP21_MOTOR_RUN 4506.07 BOOL
SEP21_OUT_DISCH_SEQ_NO D114 INT
SEP21_OUT_DISCH_SEQ_NO_INN 4705 INT
SEP21_OUT_MAIN_SEQ_NO D104 INT
SEP21_OUT_MAIN_SEQ_NO_INN 4703 INT
SEP21_OUT_MOTOR_CURR_INN 4704 REAL
SEP21_OUT_MOT_CUR_1 D106 REAL
SEP21_OUT_MOT_CUR_2 D108 DINT
SEP21_OUT_MOT_CUR_3 D110 REAL
SEP21_PRODSKUDD 4501.02 BOOL
SEP21_PRODUKT_OK 4506.03 BOOL
SEP21_RSET_FRYS T0930 BOOL
SEP21_RSET_FRYS_T 0930 NUMBER
SEP21_SEND_TIMEOUT T0800 BOOL
SEP21_SKYTER 4506.06 BOOL
SEP21_STANDBY_OK 4506.01 BOOL
SEP21_STARTET 4501.05 BOOL
SEP21_STARTET_OK 4506.00 BOOL
SEP21_START_PART_SKUDD 4504.03 BOOL  ; PAST21
SEP21_START_PRODSK 4501.08 BOOL
SEP21_STATUS_BIT 4700 INT
SEP21_STATUS_BIT_INN 4706 INT
SEP21_STOPPES 4501.13 BOOL
SEP21_STOPPSEKV_AV 4501.14 BOOL
SEP21_STOPP_SEP 4506.12 BOOL
SEP21_TOTALSKUDD 4501.04 BOOL
SEP21_UT 2400.15 BOOL
SEP21_WDOG 4506.08 BOOL
SEP21_WDOG_TIMEOUT T0801 BOOL
SEP22_0_TURTALL_FRA_SEP 1801.02 BOOL  ; SEP22 STAAR
SEP22_AUTO 1055.09 BOOL
SEP22_CIP 1800.01 BOOL  ; SEP22  C24 ER VALGT
SEP22_CIPMOD_FRA_SEP 1801.04 BOOL  ; SEP22 VASKEMODUS
SEP22_DRIFT 4511.07 BOOL
SEP22_DR_KLAR_FRA_SEP 1801.01 BOOL  ; SEP22 HAR TURTALL
SEP22_ER_SK_INTERV D3747 INT  ; INTERVALLTID SKUDD
SEP22_FEIL 4511.09 BOOL
SEP22_FEILRESET 1800.04 BOOL  ; SEP22  FEILRESET
SEP22_FEILRESET_IMP 1802.04 BOOL  ; SEP22  FEILRESET
SEP22_FEILRESET_S T0125 BOOL
SEP22_FEILRESET_T 00125 NUMBER
SEP22_FEIL_FRA_SEP 1801.08 BOOL  ; SEP22 GENERELL FEIL
SEP22_FEIL_S T0813 BOOL
SEP22_FRYSMODUS 4512.12 BOOL
SEP22_HJ_SK_INTERV D3748 INT  ; INTERVALLTID SKUDD
SEP22_INERV_START 4511.08 BOOL
SEP22_INN 2700.04 BOOL  ; SEPARATORMOTOR STARTET
SEP22_I_LINJE 4510.06 BOOL
SEP22_MAN 1005.09 BOOL
SEP22_MAN_SKUDD 4511.10 BOOL
SEP22_OK_SK_INTERV 4814.02 BOOL  ; INTERVALLTID SKUDD OK
SEP22_OWERFLOW_FRA_SEP 1801.07 BOOL  ; SEP22 SPERR UTLOEP
SEP22_P2201_MULIG_FRA_SEP 1801.00 BOOL  ; P2201 KAN STARTE
SEP22_PART_SKUDD 1800.03 BOOL  ; SEP22  START PARTIALSKUDD
SEP22_PART_SKUDD_IMP 1802.03 BOOL  ; SEP22  START PARTIALSKUDD
SEP22_PART_SKUDD_INNE_FRA_SEP 1801.05 BOOL  ; SEP22 PARTIALSKUDD
SEP22_PRODSK 4511.03 BOOL
SEP22_PRODUKT 1800.00 BOOL  ; SEP22  P2201 DRIFT
SEP22_PROD_MOD_FRA_SEP 1801.03 BOOL  ; SEP22 PRODUKTMODUS
SEP22_PRS_SK_INTERV D3746 INT  ; INTERVALLTID SKUDD
SEP22_RSET_FRYS T0931 BOOL
SEP22_SKUDD 4511.11 BOOL
SEP22_SKUDDSYKL_AV 4511.12 BOOL
SEP22_SKUDD_C D3742 INT  ; SKUDDTELLER
SEP22_SKUDD_S T0815 BOOL
SEP22_SKUDD_T 0815 NUMBER
SEP22_SK_VASK_AV 4814.01 BOOL
SEP22_SK_VASK_INN 4814.00 BOOL
SEP22_STARTET 4511.05 BOOL
SEP22_START_PART_SKUDD 4514.03 BOOL  ; PAST22
SEP22_START_PART_SKUDD_S T0124 BOOL
SEP22_START_PART_SKUDD_T 00124 NUMBER
SEP22_START_TOT_SKUDD_S T0123 BOOL
SEP22_START_TOT_SKUDD_T 00123 NUMBER
SEP22_STOPPES 4511.13 BOOL
SEP22_STOPPSEKV_AV 4511.14 BOOL
SEP22_STOPPTID_S T0814 BOOL
SEP22_SURT 1800.05 BOOL
SEP22_TOTSK 4511.04 BOOL
SEP22_TOTSK_C D3740 INT  ; ¨
SEP22_TOT_SKUDD 1800.02 BOOL  ; SEP22  START TOTALSKUDD
SEP22_TOT_SKUDD_IMP 1802.02 BOOL  ; SEP22  START TOTALSKUDD
SEP22_TOT_SKUDD_INNE_FRA_SEP 1801.06 BOOL  ; SEP22 TOTALSKUDD(VASK)
SEP22_UT 2400.04 BOOL  ; START SEPARATORMOTOR
SEP22_VIBROFEIL_1_FRA_SEP 1801.09 BOOL  ; SEP22 VIBRASJONSVARSEL. TIDLIGVARSEL
SEP22_VIBROFEIL_2_FRA_SEP 1801.10 BOOL  ; SEP22 VIBRASJONSVARSEL. SISTE VARSEL
SEP22_V_FAS_RESTTID_C D3744 INT  ; RESTID I AKTUELLE C_FASER FOR SKUDD
SEP23_START_PART_SKUDD 4524.03 BOOL  ; PAST23
SEP23_START_TOT_SKUDD 4524.02 BOOL  ; PAST21
SIGN_VACUUM 5631.06 BOOL
SIGN_VACUUM_HJ 960.05 BOOL
SIGN_VACUUM_N5 2870.04 BOOL
SILO_L3_KOEES 324.14 BOOL  ; SPERR INNLESNING TIL KOE-REGISTER.
SILO_L3_KOEPLASS_1 D5240 CHANNEL  ; XFOERST I KOE
SILO_L3_KOEPLASS_2 D5242 CHANNEL  ; X
SILO_L3_KOEPLASS_3 D5244 CHANNEL  ; X
SILO_L3_KOMMANDO_KOE 324.15 BOOL  ; D3000 VERDI KAN OVERFOERES TIL KOE-REGISTER.
SILO_L3_PAST_0_STATUS 524.01 BOOL  ; Alle objekter som ikke betjenes er ok
SILO_L3_PAST_1_STATUS 524.02 BOOL  ; Alle utstyrte objekter i 1.fase er ok
SILO_L3_PAST_2_STAT 524.03 BOOL  ; Alle utstyrte objekter er ok. Pgm = ok.
SILO_L3_PAST_DRIFT 524.00 BOOL
SILO_L3_PAST_FEIL 524.04 BOOL  ; Feil
SILO_L3_PAST_FEILTID 524.05 BOOL
SILO_L3_PAST_INDIVID_INNE 524.15 BOOL  ; Individadresse er
SILO_L3_PAST_INDKON 524.06 BOOL  ; Kontr. at bare en individadresse er hoey.
SILO_L3_PAST_OFF_IMP 524.14 BOOL
SILO_L3_PAST_ONIMPULS 524.11 BOOL  ; Startimpuls for  program
SILO_L3_PAST_RESET 524.09 BOOL  ; Stopp og nedkobling av programmet
SILO_L3_PAST_START 524.07 BOOL  ; program starter
SILO_L3_PAST_STARTIMPULS 524.10 BOOL  ; Startimpuls.
SILO_L3_TID_S T0524 BOOL  ; X
SILO_L3_TMU 524.08 BOOL
SILO_L3_TMU_TID_S T0724 BOOL  ; INKOBLINGSTID TMU NAAR LINJE IKKE AKTIVERES
SILO_L3_TMU_TID_T 0724 NUMBER  ; MAX-TID TMU OM IKKE LINJE LEGGES
SILO_L4_KOEES 325.14 BOOL  ; SPERR INNLESNING TIL KOE-REGISTER.
SILO_L4_KOEPLASS_1 D5250 CHANNEL  ; XFOERST I KOE
SILO_L4_KOEPLASS_2 D5252 CHANNEL  ; X
SILO_L4_KOEPLASS_3 D5254 CHANNEL  ; X
SILO_L4_KOMMANDO_KOE 325.15 BOOL  ; D3000 VERDI KAN OVERFOERES TIL KOE-REGISTER.
SILO_L4_PAST_0_STATUS 525.01 BOOL  ; Alle objekter som ikke betjenes er ok
SILO_L4_PAST_1_STATUS 525.02 BOOL  ; Alle utstyrte objekter i 1.fase er ok
SILO_L4_PAST_2_STAT 525.03 BOOL  ; Alle utstyrte objekter er ok. Pgm = ok.
SILO_L4_PAST_DRIFT 525.00 BOOL
SILO_L4_PAST_FEIL 525.04 BOOL  ; Feil
SILO_L4_PAST_FEILTID 525.05 BOOL
SILO_L4_PAST_INDIVID_INNE 525.15 BOOL  ; Individadresse er
SILO_L4_PAST_INDKON 525.06 BOOL  ; Kontr. at bare en individadresse er hoey.
SILO_L4_PAST_OFF_IMP 525.14 BOOL
SILO_L4_PAST_ONIMPULS 525.11 BOOL  ; Startimpuls for  program
SILO_L4_PAST_RESET 525.09 BOOL  ; Stopp og nedkobling av programmet
SILO_L4_PAST_START 525.07 BOOL  ; program starter
SILO_L4_PAST_STARTIMPULS 525.10 BOOL  ; Startimpuls.
SILO_L4_TID_S T0525 BOOL  ; X
SILO_L4_TMU 525.08 BOOL
SILO_L4_TMU_TID_S T0725 BOOL  ; INKOBLINGSTID TMU NAAR LINJE IKKE AKTIVERES
SILO_L4_TMU_TID_T 0725 NUMBER  ; MAX-TID TMU OM IKKE LINJE LEGGES
SILO_PAST21_0_STATUS 526.01 BOOL  ; Alle objekter som ikke betjenes er ok
SILO_PAST21_1_STATUS 526.02 BOOL  ; Alle utstyrte objekter i 1.fase er ok
SILO_PAST21_2_STAT 526.03 BOOL  ; Alle utstyrte objekter er ok. Pgm = ok.
SILO_PAST21_DRIFT 526.00 BOOL
SILO_PAST21_FEIL 526.04 BOOL  ; Feil
SILO_PAST21_FEILTID 526.05 BOOL
SILO_PAST21_INDIVID_INNE 526.15 BOOL  ; Individadresse er
SILO_PAST21_INDKON 526.06 BOOL  ; Kontr. at bare en individadresse er hoey.
SILO_PAST21_OFF_IMP 526.14 BOOL
SILO_PAST21_OK 4801.03 BOOL  ; LINJER FRA SILO TIL  PAST21 ER OK
SILO_PAST21_ONIMPULS 526.11 BOOL  ; Startimpuls for  program
SILO_PAST21_RESET 526.09 BOOL  ; Stopp og nedkobling av programmet
SILO_PAST21_START 526.07 BOOL  ; program starter
SILO_PAST21_STARTIMPULS 526.10 BOOL  ; Startimpuls.
SILO_PAST21_TMU 526.08 BOOL  ; Hoey bare i foerste syklus av programmet.
SILO_PAST22_0_STATUS 527.01 BOOL  ; Alle objekter som ikke betjenes er ok
SILO_PAST22_1_STATUS 527.02 BOOL  ; Alle utstyrte objekter i 1.fase er ok
SILO_PAST22_2_STAT 527.03 BOOL  ; Alle utstyrte objekter er ok. Pgm = ok.
SILO_PAST22_DRIFT 527.00 BOOL
SILO_PAST22_FEIL 527.04 BOOL  ; Feil
SILO_PAST22_FEILTID 527.05 BOOL
SILO_PAST22_INDIVID_INNE 527.15 BOOL  ; Individadresse er
SILO_PAST22_INDKON 527.06 BOOL  ; Kontr. at bare en individadresse er hoey.
SILO_PAST22_OFF_IMP 527.14 BOOL
SILO_PAST22_OK 4811.03 BOOL  ; LINJER FRA SILO TIL  PAST22 ER OK
SILO_PAST22_ONIMPULS 527.11 BOOL  ; Startimpuls for  program
SILO_PAST22_RESET 527.09 BOOL  ; Stopp og nedkobling av programmet
SILO_PAST22_START 527.07 BOOL  ; program starter
SILO_PAST22_STARTIMPULS 527.10 BOOL  ; Startimpuls.
SILO_PAST22_TMU 527.08 BOOL  ; Hoey bare i foerste syklus av programmet.
SILO_PAST23_0_STATUS 528.01 BOOL  ; Alle objekter som ikke betjenes er ok
SILO_PAST23_1_STATUS 528.02 BOOL  ; Alle utstyrte objekter i 1.fase er ok
SILO_PAST23_2_STAT 528.03 BOOL  ; Alle utstyrte objekter er ok. Pgm = ok.
SILO_PAST23_DRIFT 528.00 BOOL
SILO_PAST23_FEIL 528.04 BOOL  ; Feil
SILO_PAST23_FEILTID 528.05 BOOL
SILO_PAST23_INDIVID_INNE 528.15 BOOL  ; Individadresse er
SILO_PAST23_INDKON 528.06 BOOL  ; Kontr. at bare en individadresse er hoey.
SILO_PAST23_OFF_IMP 528.14 BOOL
SILO_PAST23_ONIMPULS 528.11 BOOL  ; Startimpuls for  program
SILO_PAST23_RESET 528.09 BOOL  ; Stopp og nedkobling av programmet
SILO_PAST23_START 528.07 BOOL  ; program starter
SILO_PAST23_STARTIMPULS 528.10 BOOL  ; Startimpuls.
SILO_PAST23_TMU 528.08 BOOL
SJELD_LAB 960.01 BOOL
SKALER_NIV_T6 D7000 REAL
SKYLL_FRA_2036 2915.14 BOOL
SKYLL_FRA_2037 2915.15 BOOL
SLC500NY_PRODKLAR_N5 2807.04 BOOL  ; FRA SLC
SLC500NY_VASKEKLAR_N5 2807.05 BOOL  ; FRA SLC
SLC500NY_VASKELOEP_OK_N5 2807.06 BOOL  ; FRA SLC
SLC500_C45_INNE_PR2 5010.02 BOOL  ; VASK C45 ER I DRIFT
SLC500_LUT_PR2 5117.02 BOOL  ; DOSER LUT FRA P8007
SLC500_PRODUKSJON_N5 2802.01 BOOL  ; SLC ER KLAR TIL PRODUKSJON
SLC500_PROD_PR2 5117.05 BOOL  ; SLC ER KLAR TIL PRODUKSJON
SLC500_PR_INNE_PR2 5010.03 BOOL  ; PRODUKT FRA T20.11 TIL 20.19 ER INNKOBLET
SLC500_SYRE_PR2 5117.03 BOOL  ; DOSER SYRET FRA P8008
SLC500_VASK_N5 2802.00 BOOL  ; SLC ER KLAR TIL VASK
SLC500_VASK_PR2 5117.04 BOOL  ; SLC ER KLAR TIL VASK
SPANN_D_FOR 723.11 BOOL  ; FRA CONTAINER(SPANN) TIL T27.40-41
SPANN_D_FOR_COM_BIT 1150.01 BOOL  ; TIL T27.40-41.
SPERR_RV_MELK_T2036 925.00 BOOL  ; Bitt settes i InTouch for aa unngaa at roereverk starter automatisk dersom det er ren melk paa tanken.
SPERR_RV_MELK_T2037 925.01 BOOL  ; Bitt settes i InTouch for aa unngaa at roereverk starter automatisk dersom det er ren melk paa tanken.
SPERR_T81 1401.00 BOOL  ; Sperr Tank 81. Forskylletank.
SPERR_T82 1402.00 BOOL  ; Sperr Tank 82. Luttank.
SPERR_T83 1403.00 BOOL  ; Sperr Tank 83. Syretank.
SPERR_T84 1404.00 BOOL  ; Sperr Tank 84. Hetvanntank.
SPJELD_LAB 960.01 BOOL
STARTP_DREN_L11 712.09 BOOL
STARTP_DREN_L12 714.09 BOOL
STARTP_DREN_L21 716.09 BOOL
STARTP_DREN_L22 718.09 BOOL
STARTST_V4302_N5 2824.00 BOOL
START_MD_L11_S T0664 BOOL
START_MD_L12_S T0665 BOOL
START_MD_L21_S T0666 BOOL
START_MD_L22_S T0667 BOOL
START_PROFIBUS_UNIT1 1525.00 BOOL  ; STARTBIT=1500+(25*UNITNR).01
START_PROFIBUS_UNIT2 1550.00 BOOL  ; STARTBIT=1500+(25*UNITNR).02
START_PROFIBUS_UNIT3 1575.00 BOOL  ; STARTBIT=1500+(25*UNITNR).03
START_PROFIBUS_UNIT5 1625.00 BOOL  ; STARTBIT=1500+(25*UNITNR).05
START_V4302 2561.10 BOOL
START_VD_L11_S T0660 BOOL
START_VD_L12_S T0661 BOOL
START_VD_L21_S T0662 BOOL
START_VD_L22_S T0663 BOOL
STOPP_SIRK_T82 1406.00 BOOL
SUM_LINJEFEIL 999.05 BOOL
S_8019 2505.04 BOOL  ; VST80-K1-RETUR TIL GRM.
T03_520_1_HJ1 936.06 BOOL
T03_520_1_HJ2 936.07 BOOL
T03_521_1_HJ1 936.13 BOOL
T03_521_1_HJ2 936.14 BOOL
T03_522_1_HJ1 937.04 BOOL
T03_522_1_HJ2 937.05 BOOL
T03_523_1_HJ1 937.11 BOOL
T03_523_1_HJ2 937.12 BOOL
T03_524_1_HJ1 938.02 BOOL
T03_524_1_HJ2 938.03 BOOL
T03_525_1_HJ1 938.09 BOOL
T03_525_1_HJ2 938.10 BOOL
T03_FRA_L1_MELK 601.01 BOOL
T03_FRA_L1_MELK_HR H60.01 BOOL  ; HUSKER STATUS
T03_FRA_L1_VANN 601.00 BOOL
T03_FRA_L1_VANN_HR H60.00 BOOL  ; HUSKER STATUS
T03_FRA_L2_MELK 601.04 BOOL
T03_FRA_L2_MELK_HR H60.03 BOOL  ; HUSKER STATUS
T03_FRA_L2_VANN 601.03 BOOL
T03_FRA_L2_VANN_HR H60.02 BOOL  ; HUSKER STATUS
T03_HL 2600.12 BOOL  ; Z
T03_L2_DREN_1_ST 601.11 BOOL  ; FRA V0339
T03_L3_PAST_IND 1224.00 BOOL  ; TIL PASTEURER VIA LINJE 3
T03_L3_VALG 324.00 BOOL  ; INDIVIDVALG FRA KOEREGISTER.
T03_L4_PAST_IND 1225.00 BOOL  ; INDIVIDADRESSE.
T03_L4_VALG 325.00 BOOL  ; INDIVIDVALG FRA KOEREGISTER.
T03_LINJETOEM_VASK 601.12 BOOL  ; V0310-20-30-40 NEDRE VASKELOEP AAPNES ETTER VASK
T03_LINJETOEM_VASK_S C0063 BOOL  ; AAPNINGSTID NAAR V0310-20-30-40 NEDRE VASKELOEP AAPNES ETTER VASK
T03_LINJETOEM_VASK_T C63 CHANNEL  ; AAPNINGSTID NAAR V0310-20-30-40 NEDRE VASKELOEP AAPNES ETTER VASK
T03_LL_PRS_TID D6004 WORD  ; PRS TID FOR LL T03
T03_RV0301_DRIFT_HR H60.08 BOOL
T03_SIST_FRA_L1 600.12 BOOL
T03_SIST_FRA_L1_1 600.08 BOOL
T03_SIST_FRA_L1_2 600.09 BOOL
T03_SIST_FRA_L2 600.13 BOOL
T03_SIST_FRA_L2_1 600.10 BOOL
T03_SIST_FRA_L2_2 600.11 BOOL
T03_SPERR 601.15 BOOL  ; SPERRER ALLE FUNKSJONER TIL/ FRA TANK. OGSAA VASK
T03_SPERRET_HR H60.07 BOOL
T03_SPERR_KODE_INN D6008 CHANNEL
T03_SPERR_KODE_UT D6009 CHANNEL
T03_TANKTOEM_VASK 601.13 BOOL  ; V0306-08-71AAPNES ETTER VASK
T03_TANKTOEM_VASK_S C0069 BOOL  ; AAPNINGSTID TIL SLUK ETTER TANKVASK
T03_TANKTOEM_VASK_T C69 CHANNEL  ; AAPNINGSTID TIL SLUK ETTER TANKVASK
T03_TL1_DRENER 600.14 BOOL  ; FRA V329
T03_TL1_DRENSTID_S T0037 BOOL
T03_TL1_DRENSTID_T 0037 NUMBER
T03_TL1_DREN_1_ST 601.09 BOOL  ; FRA V0329
T03_TL1_ROER_VASKET 601.07 BOOL
T03_TL1_ROER_VASKET_HR H60.05 BOOL  ; HUSKER STATUS
T03_TL2_DRENER 600.15 BOOL  ; FRA V339
T03_TL2_DRENSTID_S T0038 BOOL
T03_TL2_DRENSTID_T 0038 NUMBER
T03_TL2_ROER_VASKET 601.08 BOOL
T03_TL2_ROER_VASKET_HR H60.06 BOOL
T03_VASKET 601.06 BOOL
T03_VASKET_4 H60.04 BOOL  ; HUSKER STATUS
T04_520_1_HJ1 936.08 BOOL
T04_520_1_HJ2 936.09 BOOL
T04_521_1_HJ1 936.15 BOOL
T04_521_1_HJ2 937.00 BOOL
T04_522_1_HJ1 937.06 BOOL
T04_522_1_HJ2 937.07 BOOL
T04_523_1_HJ1 937.13 BOOL
T04_523_1_HJ2 937.14 BOOL
T04_524_1_HJ1 938.04 BOOL
T04_524_1_HJ2 938.05 BOOL
T04_525_1_HJ1 938.11 BOOL
T04_525_1_HJ2 938.12 BOOL
T04_FRA_L1_MELK 603.01 BOOL
T04_FRA_L1_MELK_HR H62.01 BOOL  ; HUSKER STATUS
T04_FRA_L1_VANN 603.00 BOOL
T04_FRA_L1_VANN_HR H62.00 BOOL  ; HUSKER STATUS
T04_FRA_L2_MELK 603.04 BOOL
T04_FRA_L2_MELK_HR H62.03 BOOL  ; HUSKER STATUS
T04_FRA_L2_VANN 603.03 BOOL
T04_FRA_L2_VANN_HR H62.02 BOOL  ; HUSKER STATUS
T04_L1_DREN_1_ST 603.09 BOOL  ; FRA V0429
T04_L2_DREN_1_ST 603.11 BOOL  ; FRA V0439
T04_L3_PAST_IND 1224.01 BOOL  ; TIL PASTEURER VIA LINJE 3
T04_L3_VALG 324.01 BOOL  ; INDIVIDVALG FRA KOEREGISTER.
T04_L4_PAST_IND 1225.01 BOOL  ; INDIVIDADRESSE.
T04_L4_VALG 325.01 BOOL  ; INDIVIDVALG FRA KOEREGISTER.
T04_LINJETOEM_VASK 603.12 BOOL  ; V0410-20-30-40 NEDRE VASKELOEP AAPNES ETTER VASK
T04_LINJETOEM_VASK_S C0064 BOOL  ; AAPNINGSTID NAAR V0410-20-30-40 NEDRE VASKELOEP AAPNES ETTER VASK
T04_LINJETOEM_VASK_T C64 CHANNEL  ; AAPNINGSTID NAAR V0410-20-30-40 NEDRE VASKELOEP AAPNES ETTER VASK
T04_LL_F0RSINKELSE C0621 BOOL  ; FORSINKER INNKOBLING AV BUNNSIGNAL
T04_LL_PRS_TID D6024 WORD  ; PRS TID FOR LL T04
T04_MIDL_SPERRE 999.09 BOOL
T04_RV0401_DRIFT_HR H62.08 BOOL
T04_RV0402_DRIFT_HR H62.09 BOOL
T04_SIST_FRA_L1 602.12 BOOL
T04_SIST_FRA_L1_1 602.08 BOOL
T04_SIST_FRA_L1_2 602.09 BOOL
T04_SIST_FRA_L2 602.13 BOOL
T04_SIST_FRA_L2_1 602.10 BOOL
T04_SIST_FRA_L2_2 602.11 BOOL
T04_SPERR 603.15 BOOL  ; SPERRER ALLE FUNKSJONER TIL/ FRA TANK. OGSAA VASK
T04_SPERRET_HR H62.07 BOOL
T04_SPERR_KODE_INN D6028 CHANNEL
T04_SPERR_KODE_UT D6029 CHANNEL
T04_TANKTOEM_VASK 603.13 BOOL  ; V0406-08-71AAPNES ETTER VASK
T04_TANKTOEM_VASK_S C0070 BOOL  ; AAPNINGSTID TIL SLUK ETTER TANKVASK
T04_TANKTOEM_VASK_T C70 CHANNEL  ; AAPNINGSTID TIL SLUK ETTER TANKVASK
T04_TL1_DRENER 602.14 BOOL  ; FRA V429
T04_TL1_DRENSTID_S T0039 BOOL
T04_TL1_DRENSTID_T 0039 NUMBER
T04_TL1_ROER_VASKET 603.07 BOOL
T04_TL1_ROER_VASKET_HR H62.05 BOOL  ; HUSKER STATUS
T04_TL2_DRENER 602.15 BOOL  ; FRA V439
T04_TL2_DRENSTID_S T0040 BOOL
T04_TL2_DRENSTID_T 0040 NUMBER
T04_TL2_ROER_VASKET 603.08 BOOL
T04_TL2_ROER_VASKET_HR H62.06 BOOL
T04_VASKET 603.06 BOOL
T04_VASKET_4 H62.04 BOOL  ; HUSKER STATUS
T05_520_1_HJ1 936.10 BOOL
T05_520_1_HJ2 936.11 BOOL
T05_521_1_HJ1 937.01 BOOL
T05_521_1_HJ2 937.02 BOOL
T05_522_1_HJ1 937.08 BOOL
T05_522_1_HJ2 937.09 BOOL
T05_523_1_HJ1 937.15 BOOL
T05_523_1_HJ2 938.00 BOOL
T05_524_1_HJ1 938.06 BOOL
T05_524_1_HJ2 938.07 BOOL
T05_525_1_HJ1 938.13 BOOL
T05_525_1_HJ2 938.14 BOOL
T05_FRA_L1_MELK 605.01 BOOL
T05_FRA_L1_MELK_HR H64.01 BOOL  ; HUSKER STATUS
T05_FRA_L1_VANN 605.00 BOOL
T05_FRA_L1_VANN_HR H64.00 BOOL  ; HUSKER STATUS
T05_FRA_L2_DRENERT 605.05 BOOL
T05_FRA_L2_MELK 605.04 BOOL
T05_FRA_L2_MELK_HR H64.03 BOOL  ; HUSKER STATUS
T05_FRA_L2_VANN 605.03 BOOL
T05_HL 2600.02 BOOL  ; HL-T05
T05_L1_DREN_1_ST 605.09 BOOL  ; FRA V0529
T05_L2_DREN_1_ST 605.11 BOOL  ; FRA V0539
T05_L3_PAST_IND 1224.02 BOOL  ; TIL PASTEURER VIA LINJE 3
T05_L3_VALG 324.02 BOOL  ; INDIVIDVALG FRA KOEREGISTER.
T05_L4_PAST_IND 1225.02 BOOL  ; INDIVIDADRESSE.
T05_L4_VALG 325.02 BOOL  ; INDIVIDVALG FRA KOEREGISTER.
T05_LINJETOEM_VASK 605.12 BOOL  ; V0510-20-30-40 NEDRE VASKELOEP AAPNES ETTER VASK
T05_LINJETOEM_VASK_S C0065 BOOL  ; AAPNINGSTID NAAR V0510-20-30-40 NEDRE VASKELOEP AAPNES ETTER VASK
T05_LINJETOEM_VASK_T C65 CHANNEL  ; AAPNINGSTID NAAR V0510-20-30-40 NEDRE VASKELOEP AAPNES ETTER VASK
T05_LL_F0RSINKELSE C0641 BOOL  ; FORSINKER INNKOBLING AV BUNNSIGNAL
T05_LL_PRS_TID D6044 WORD  ; PRS TID FOR LL T05
T05_MIDL_SP 999.10 BOOL
T05_RV0401_DRIFT_HR H64.08 BOOL
T05_RV0501_DRIFT_HR H62.10 BOOL
T05_RV0502_DRIFT_HR H62.11 BOOL
T05_SIST_FRA_L1 604.12 BOOL
T05_SIST_FRA_L1_1 604.08 BOOL
T05_SIST_FRA_L1_2 604.09 BOOL
T05_SIST_FRA_L2 604.13 BOOL
T05_SIST_FRA_L2_1 604.10 BOOL
T05_SIST_FRA_L2_2 604.11 BOOL
T05_SPERR 605.15 BOOL  ; SPERRER ALLE FUNKSJONER TIL/ FRA TANK. OGSAA VASK
T05_SPERRET_HR H64.07 BOOL
T05_SPERR_KODE_INN D6048 CHANNEL
T05_SPERR_KODE_UT D6049 CHANNEL
T05_TANKTOEM_VASK 605.13 BOOL  ; V0506-08-71AAPNES ETTER VASK
T05_TANKTOEM_VASK_S C0071 BOOL  ; AAPNINGSTID TIL SLUK ETTER TANKVASK
T05_TANKTOEM_VASK_T C71 CHANNEL  ; AAPNINGSTID TIL SLUK ETTER TANKVASK
T05_TL1_DRENER 604.14 BOOL  ; FRA V529
T05_TL1_DRENSTID_S T0041 BOOL
T05_TL1_DRENSTID_T 0041 NUMBER
T05_TL1_ROER_VASKET 605.07 BOOL
T05_TL1_ROER_VASKET_HR H64.05 BOOL  ; HUSKER STATUS
T05_TL2_DRENER 604.15 BOOL  ; FRA V539
T05_TL2_DRENSTID_S T0042 BOOL
T05_TL2_DRENSTID_T 0042 NUMBER
T05_TL2_ROER_VASKET 605.08 BOOL
T05_TL2_ROER_VASKET_HR H64.06 BOOL
T05_VASKET 605.06 BOOL
T05_VASKET_4 H64.04 BOOL  ; HUSKER STATUS
T06_AUTOSPERR_AKTIV 607.10 BOOL
T06_AUTOSPERR_AKTIVERES 607.09 BOOL
T06_AUTOSPERR_DAG D7010 INT
T06_AUTOSPERR_HJ D7014 INT
T06_AUTOSPERR_MAANED D7011 INT
T06_AUTOSPERR_MINUTT D7013 INT
T06_AUTOSPERR_TIME D7012 INT
T06_AUTOSPERR_VALGT 607.08 BOOL
T06_AUTOTOEMMING_AKTIV 607.13 BOOL
T06_AUTOTOEMMING_AKTIVERES 607.12 BOOL
T06_AUTOTOEMMING_DAG D7020 INT
T06_AUTOTOEMMING_HJ D7024 INT
T06_AUTOTOEMMING_MAANED D7021 INT
T06_AUTOTOEMMING_MINUTT D7023 INT
T06_AUTOTOEMMING_TIME D7022 INT
T06_AUTOTOEMMING_VALGT 607.11 BOOL
T06_C30_START 608.00 BOOL  ; STARTIMPULS TIL C30
T06_DR_HYDROPHOR 607.14 BOOL
T06_HL 607.00 BOOL  ; FORS.
T06_HL_S T0892 BOOL
T06_HYDROPHOR_UT 2403.03 BOOL
T06_HYDROPH_UT_PR2 5022.00 BOOL  ; FRA NODE1
T06_LL 607.01 BOOL  ; FORS.
T06_LL_S T0893 BOOL
T06_MANUELL_BYPASS_UV_LYS 607.07 BOOL
T06_MANUELL_SPERRING 607.04 BOOL
T06_MANUELL_SPERR_HYDROPHOR 607.06 BOOL
T06_MANUELL_TOEMMING 607.05 BOOL
T06_OMKOBL_NIV_HYDROPHOR 607.02 BOOL
T06_RESET_LITER 608.02 BOOL  ; RESETD6078
T06_RESET_MAX_FLOW 608.01 BOOL  ; RESET D6076
T06_SPERR 607.15 BOOL  ; SPERRER ALLE FUNKSJONER TIL/ FRA TANK. OGSAA VASK
T06_SPERRET_HR H66.07 BOOL
T06_SPERR_KODE_INN D6060 CHANNEL
T06_SPERR_KODE_UT D6061 CHANNEL
T06_VASKET 607.03 BOOL  ; C30
T0905_VASKET_N6 2828.15 BOOL
T2009_P23_PROD_ETTER_C25 4824.02 BOOL  ; FOERSTE PRODUKTKJOERING ETTER VASK
T2009_P23_PROD_ETTER_C25_S T0827 BOOL  ; FORSINKET UT 4824.02
T2009_P23_PROD_ETTER_C25_T 0827 NUMBER  ; FORSINKET UT 4824.02
T2009_P23_VANN_UT 4824.03 BOOL  ; LINJE TOEMMES FOR VANN
T2009_P23_VANN_UT_S T0825 BOOL  ; FOERSTE PRODUKTKJOERING ETTER VASK
T2009_P23_VANN_UT_T 0825 NUMBER  ; FOERSTE PRODUKTKJOERING ETTER VASK
T2011_37_MANUELL 698.02 BOOL  ; MANUELT FRAM TIL SLUK/FOR
T2011__37_MANUELL_AAPNING_N4 2936.02 BOOL  ; MANUELL AAPNING T2011-19 OG 36-37
T2036_DREN_FOR 2909.06 BOOL
T2036_DREN_SLUK 2909.07 BOOL
T2036_DREN_UHT 2909.08 BOOL
T2037_DREN_FOR 2909.09 BOOL
T2037_DREN_SLUK 2909.10 BOOL
T2037_DREN_UHT 2909.11 BOOL
T20M3_COMAND_ORD 2913 WORD  ; 1=SLUK                                                                     2=DYREFOR
T20M3_D_FOR 723.07 BOOL  ; TIL TANK TIL T27.40-41
T20M3_SLUK 723.06 BOOL
T20_11_MAN_N5 2800.12 BOOL
T20_17_HL_PR2 5117.00 BOOL
T20_17_LL_N5 2805.06 BOOL
T20_17_LL_PR2 5117.01 BOOL
T20_36_LL_N5 2909.12 BOOL
T20_36_MAN_N5 2805.00 BOOL
T20_36_SPERR_N1 411.12 BOOL
T20_37_LL_N5 2909.13 BOOL
T20_37_MAN_N5 2805.01 BOOL
T20_37_SPERR_N5 2800.13 BOOL
T22_SURT_UT_22GR 4814.09 BOOL
T24_01_KLAR_TIL_VASKES 750.04 BOOL
T24_01_PRODUKT 750.03 BOOL
T24_01_SPERR 750.02 BOOL  ; SPERRER ALLE FUNKSJONER TIL/ FRA TANK. OGSAA VASK
T24_01_SPERRET_HR H60.11 BOOL
T24_01_VASKES 750.05 BOOL
T24_01_VASKET 750.06 BOOL
T24_SPERR_KODE_INN D6244 CHANNEL
T24_SPERR_KODE_UT D6245 CHANNEL
T25M3_COMAND_ORD 2910 WORD  ; 1=SLUK                                                                     2=DYREFOR
T25M3_D_FOR 723.01 BOOL  ; TIL TANK TIL T27.40-41
T25M3_SLUK 723.00 BOOL
T2701_BIL_DRENERER 544.13 BOOL
T2701_BIL_DRENSTID_S T0890 BOOL
T2701_BIL_DRENSTID_SLUK_S T0891 BOOL
T2701_BIL_DREN_UTFOERT 688.13 BOOL
T2701_BIL_MELK 688.11 BOOL
T2701_BIL_TOEMMER 544.12 BOOL
T2701_KAN_VASKES 688.04 BOOL
T2701_PRODUKT 688.03 BOOL
T2701_PT D6092 INT  ; T2701-OEKOMELK
T2701_SPERR 688.02 BOOL  ; SPERRER ALLE FUNKSJONER TIL/ FRA TANK. OGSAA VASK
T2701_SPERRET_HR H60.12 BOOL
T2701_SPERR_KODE_INN D6246 CHANNEL
T2701_SPERR_KODE_UT D6247 CHANNEL
T2701_TT D6090 INT  ; T2701-OEKOMELK
T2701_VASKES 688.05 BOOL
T2701_VASKET 688.06 BOOL
T2702_KAN_VASKES 689.04 BOOL
T2702_PRODUKT 689.03 BOOL
T2702_PT D6094 INT  ; T2702-RETURMELK
T2702_SPERR 689.02 BOOL  ; SPERRER ALLE FUNKSJONER TIL/ FRA TANK. OGSAA VASK
T2702_SPERRET_HR H60.13 BOOL
T2702_SPERR_KODE_INN D6248 CHANNEL
T2702_SPERR_KODE_UT D6249 CHANNEL
T2702_VASKES 689.05 BOOL
T2702_VASKET 689.06 BOOL
T2703_KAN_VASKES 690.04 BOOL
T2703_PRODUKT 690.03 BOOL
T2703_PT D6096 INT  ; T2703-RETURMELK
T2703_SPERR 690.02 BOOL  ; ¨
T2703_SPERRET_HR H60.14 BOOL
T2703_SPERR_KODE_INN D6250 CHANNEL
T2703_SPERR_KODE_UT D6251 CHANNEL
T2703_VASKES 690.05 BOOL
T2703_VASKET 690.06 BOOL
T27_01_HL_FORSINKELSE_S T0896 BOOL  ; TID SOM FORSINKER  TOPPVARSEL PAA T24.01
T27_01_LL_FORSINKELSE_S T0897 BOOL  ; TID SOM FORSINKER   BUNNVARSEL PAA T27.01
T27_02_HL_FORSINKELSE_S T0898 BOOL  ; TID SOM FORSINKER  TOPPVARSEL PAA  TANK
T27_02_LL_FORSINKELSE_S T0899 BOOL  ; TID SOM FORSINKER   BUNNVARSEL PAA TANK
T27_03_HL_FORSINKELSE_S T0900 BOOL  ; TID SOM FORSINKER  TOPPVARSEL PAA  TANK
T27_03_LL_FORSINKELSE_S T0901 BOOL  ; TID SOM FORSINKER   BUNNVARSEL PAA TANK
T40_KAN_VASKES 648.04 BOOL
T40_PRODUKT 648.03 BOOL
T40_SKYLL_AVSL 648.15 BOOL
T40_SKYLL_START 648.14 BOOL
T40_SKYLL_TID_S T1002 BOOL
T40_SKYLL_TID_T 1002 NUMBER
T40_SPERR 648.02 BOOL  ; SPERRER ALLE FUNKSJONER TIL/ FRA TANK. OGSAA VASK
T40_SPERRET_HR H60.09 BOOL
T40_SPERR_KODE_INN D6240 CHANNEL
T40_SPERR_KODE_UT D6241 CHANNEL
T40_VASKES 648.05 BOOL
T40_VASKET 648.06 BOOL
T41_KAN_VASKES 649.04 BOOL
T41_PRODUKT 649.03 BOOL
T41_SKYLL_AVSL 649.15 BOOL
T41_SKYLL_START 649.14 BOOL
T41_SKYLL_TID_S T1003 BOOL
T41_SKYLL_TID_T 1003 NUMBER
T41_SPERR 649.02 BOOL  ; SPERRER ALLE FUNKSJONER TIL/ FRA TANK. OGSAA VASK
T41_SPERRET_HR H60.10 BOOL
T41_SPERR_KODE_INN D6242 CHANNEL
T41_SPERR_KODE_UT D6243 CHANNEL
T41_VASKES 649.05 BOOL
T41_VASKET 649.06 BOOL
T7M3_COMAND_ORD 2912 WORD  ; 1=SLUK                                                                     2=DYREFOR
T7M3_D_FOR 723.05 BOOL  ; TIL TANK TIL T27.40-41
T7M3_SLUK 723.04 BOOL
T81_FEIL 1401.12 BOOL
T81_FEILBETING 1401.13 BOOL  ; FEILBETINGELSER
T81_HL 2501.12 BOOL  ; VST80_T82_FORS_TANK
T81_HL_TID T0016 BOOL
T81_INTERN_SIRK 1401.15 BOOL  ; T81  INTERN SIRKULASJON BENYTTES VED INTERNVASK AV VASKESTASJONEN
T81_LL_TID T0017 BOOL
T81_NIVAA D8108 CHANNEL
T81_NIV_HJF1 900.00 BOOL
T81_SPERR_HR H1.04 BOOL  ; RETENTETIV FUNKSJON
T81_SPERR_KODE_INN D8110 CHANNEL
T81_SPERR_KODE_UT D8111 CHANNEL
T81_TEMP_HOY 1401.14 BOOL  ; T81 TANKTEMP FOR HOEY
T82_CT_HJ1 900.04 BOOL
T82_DOS_TID_S T0105 BOOL  ; T82 DOSERINGSTID LUT
T82_ERV_KOND D8200 CHANNEL
T82_ER_TEMP D8204 CHANNEL
T82_FEIL 1402.12 BOOL
T82_FEIL_HJ_CON 900.07 BOOL  ; MIN-COND. FOER ALARM
T82_FEIL_HJ_NIV 900.06 BOOL
T82_HL 2501.13 BOOL  ; VST80_T82_LUTTANK
T82_HL_TID T0018 BOOL
T82_HYST_COND D8222 CHANNEL
T82_HYST_TEMP D8224 CHANNEL
T82_INTERN_SIRK 1402.15 BOOL  ; T82  INTERN SIRKULASJON BENYTTES VED INTERNVASK AV VASKESTASJONEN
T82_KONDLAV_KURSKONTR 1402.09 BOOL  ; FOR LAV KONSENTRASJON PAA TANK TIL AA STARTE LUTFASE.
T82_KURS_CONDKONTR D8232 CHANNEL  ; FOR LAV KONSENTRASJON PAA TANK TIL AA STARTE LUTFASE.
T82_LL_TID T0019 BOOL
T82_MAN_DOS_TID T0072 BOOL  ; MAXTID MANUELL DOSERING KAN VAERE INNE PR GANG
T82_MAN_DOS_TID_T 0072 NUMBER  ; MAXTID MANUELL DOSERING KAN VAERE INNE PR GANG
T82_MIN_COND D8228 CHANNEL  ; MINIMUMSKOND. FOER ALARM
T82_MIN_TEMP D8230 CHANNEL  ; MINIMUMSTEMP FOER ALARM
T82_NEDRE_TEMP D8226 INT
T82_NIVAA D8208 CHANNEL
T82_NIV_HJF1 900.01 BOOL
T82_OPPVARM_OK T0181 BOOL
T82_OPPV_OK D8242 INT
T82_PAUSE_TID_S T0106 BOOL  ; T82 PAUSETID LUT-DOSERING
T82_PRS_COND D8202 CHANNEL
T82_SPERR_HR H1.05 BOOL  ; RETENTETIV FUNKSJON
T82_SPERR_KODE_INN D8210 CHANNEL
T82_SPERR_KODE_UT D8211 CHANNEL
T82_START_OPPV D8240 INT
T83_CT_HJ1 900.05 BOOL
T83_DOS_TID_S T0107 BOOL  ; T83 DOSERINGSTID LUT
T83_ERV_KOND D8300 CHANNEL
T83_ER_TEMP D8304 CHANNEL
T83_FEIL 1403.12 BOOL
T83_FEIL_HJ_CON 900.09 BOOL  ; MIN-COND. FOER ALARM
T83_FEIL_HJ_NIV 900.08 BOOL
T83_HL 2501.14 BOOL  ; VST80_T83_SYRETANK
T83_HL_TID T0020 BOOL
T83_HYST_COND D8322 CHANNEL
T83_HYST_TEMP D8324 CHANNEL
T83_INTERN_SIRK 1403.15 BOOL  ; T83  INTERN SIRKULASJON BENYTTES VED INTERNVASK AV VASKESTASJONEN
T83_LL_TID T0021 BOOL
T83_MAN_DOS_TID T0073 BOOL  ; MAXTID MANUELL DOSERING KAN VAERE INNE PR GANG
T83_MAN_DOS_TID_T 0073 NUMBER  ; MAXTID MANUELL DOSERING KAN VAERE INNE PR GANG
T83_MIN_COND D8328 CHANNEL  ; MINIMUMSKONDUKTIVITET FOER ALARM
T83_MIN_TEMP D8330 CHANNEL  ; MINIMUMSTEMP FOER ALARM
T83_NEDRE_TEMP D8326 INT
T83_NIVAA D8308 CHANNEL
T83_NIV_HJF1 900.02 BOOL
T83_PAUSE_TID_S T0108 BOOL  ; T83 PAUSETID LUT-DOSERING
T83_PRS_COND D8302 CHANNEL
T83_SPERR_HR H1.06 BOOL  ; RETENTETIV FUNKSJON
T83_SPERR_KODE_INN D8310 CHANNEL
T83_SPERR_KODE_UT D8311 CHANNEL
T83_TEMP_PRS D8306 INT
T84_CT_HJ1 900.11 BOOL
T84_C_N_DOS_BR_PR2_06 5113.00 BOOL  ; FRA PROFIBUS                                                   BRYTER  NOEDOSERING T84
T84_C_N_DOS_LA_PR2_06 5008.00 BOOL
T84_DOS_TID_S T0112 BOOL
T84_ERV_COND D8400 INT
T84_ER_TEMP D8404 CHANNEL
T84_FEIL 1404.12 BOOL
T84_FEIL_HJ_NIV 900.10 BOOL
T84_HL 2501.15 BOOL  ; VST80_T84_HETV_TANK
T84_HL_TID T0022 BOOL
T84_HL_T_V8420_S T0119 BOOL
T84_HYST_COND D8422 INT
T84_INTERN_SIRK 1404.15 BOOL  ; T83  INTERN SIRKULASJON BENYTTES VED INTERNVASK AV VASKESTASJONEN
T84_KONDLAV_KURSKONTR 1404.09 BOOL  ; FOR LAV KONSENTRASJON PAA TANK TIL AA STARTE LUTFASE.
T84_KURS_CONDKONTR D8432 CHANNEL  ; FOR LAV KONSENTRASJON PAA TANK TIL AA STARTE LUTFASE.
T84_LL_TID T0023 BOOL
T84_MAN_DOS_TID T0074 BOOL  ; MAXTID MANUELL DOSERING KAN VAERE INNE PR GANG
T84_MAN_DOS_TID_T 0074 NUMBER  ; MAXTID MANUELL DOSERING KAN VAERE INNE PR GANG
T84_NIVAA D8408 CHANNEL
T84_NIV_HJF1 900.03 BOOL
T84_PAUSE_TID_S T0113 BOOL
T84_PRS_COND D8402 INT
T84_SPERR_HR H1.07 BOOL  ; RETENTETIV FUNKSJON
T84_SPERR_KODE_INN D8410 CHANNEL
T84_SPERR_KODE_UT D8411 CHANNEL
T8M3_COMAND_ORD 2911 WORD  ; 1=SLUK                                                                     2=DYREFOR
T8M3_D_FOR 723.03 BOOL  ; TIL TANK TIL T27.40-41
T8M3_SLUK 723.02 BOOL
TEMP_MAX_K1 D9704 INT
TEMP_MAX_K2 D9706 INT
TEMP_MAX_K3 D9708 INT
TID_V_8001 T0013 BOOL
TID_V_8002 100.14 BOOL
TID_V_8002_ T0014 BOOL
TID_V_8003 T0015 BOOL
TIL_N5_C79_IND 2805.14 BOOL
TOT_MENG_MOT_RESET 698.05 BOOL  ; RESETTER TOTALTELLERNE I MOTTAK
TRAKT_SLUK 723.10 BOOL  ; TRAKT TIL SLUK
TRAKT_SLUK_COM_BIT 1150.00 BOOL  ; TRAKT TIL SLUK
TRINN_HOMOTR1_S T0002 BOOL
TR_L1_1_C81_CONTAINER 1309.05 BOOL  ; KNAPP PAA VEGG VED L1.2 FOR AA VELGE C81 SOM CONTAINERVASK
TR_L1_1_C81_CONTAINER_S T0912 BOOL
TR_L1_2_C81_CONTEINER 2603.09 BOOL  ; TR.KNAPP PAA VEGG VED L1.2 FOR VALG AV CONTAINERVASK VIA C81
T_VENTILF_SIRK_K1 T0005 BOOL
T_VENTILF_SIRK_K2 T0006 BOOL
T_VENTILF_SIRK_K3 T0007 BOOL
UTG_P8001 5474 CHANNEL
UTG_P8002 5475 CHANNEL
V0101_INN 2519.00 BOOL  ; Z
V0101_UT 2219.00 BOOL  ; Z
V0104_INN 2519.03 BOOL  ; Z
V0104_INN_FORS_S T0080 BOOL
V0104_INN_FORS_T 080 NUMBER
V0104_LINJE_INAKTIV 701.12 BOOL  ; VENTIL STENGT. INGEN AKTIVITET PAA L1.1
V0104_LINJE_INAKTIV_S C0131 BOOL  ; VENTIL STENGT. INGEN AKTIVITET PAA L1.1
V0104_LINJE_INAKTIV_T C131 CHANNEL  ; VENTIL STENGT. INGEN AKTIVITET PAA L1.1
V0104_STENGER 700.14 BOOL
V0104_UT 2219.03 BOOL  ; Z
V0104_UT_FORS_S T0081 BOOL
V0104_UT_FORS_T 081 NUMBER
V0104_UT_ML_FORS_S T0075 BOOL
V0104_UT_ML_FORS_T 075 NUMBER
V0105_INN 2519.04 BOOL  ; Z
V0105_UT 2219.04 BOOL  ; Z
V0106_INN 2519.12 BOOL  ; Z
V0106_UT 2219.12 BOOL  ; Z
V0107_INN 2519.05 BOOL  ; Z
V0107_UT 2219.05 BOOL  ; Z
V0108_INN 2519.13 BOOL  ; Z
V0108_UT 2219.13 BOOL  ; Z
V0109_INN 2515.04 BOOL  ; Z
V0109_UT 2215.04 BOOL  ; Z
V0110_INN 2519.15 BOOL  ; Z
V0110_UT 2219.15 BOOL  ; Z
V0111_INN 2519.07 BOOL  ; Z
V0111_UT 2219.07 BOOL  ; Z
V0114_INN 2519.10 BOOL  ; Z
V0114_INN_FORS_S T0085 BOOL
V0114_INN_FORS_T 085 NUMBER
V0114_LINJE_INAKTIV_S C0132 BOOL  ; VENTIL STENGT. INGEN AKTIVITET PAA L1.2
V0114_LINJE_INAKTIV_T C132 CHANNEL  ; VENTIL STENGT. INGEN AKTIVITET PAA L1.2
V0114_STENGER 702.14 BOOL
V0114_UT 2219.10 BOOL  ; Z
V0114_UT_FORS_S T0086 BOOL
V0114_UT_FORS_T 086 NUMBER
V0114_UT_ML_FORS_S T0076 BOOL
V0114_UT_ML_FORS_T 076 NUMBER
V0115_INN 2519.11 BOOL  ; Z
V0115_UT 2219.11 BOOL  ; Z
V0117_INN 2515.03 BOOL  ; Z
V0117_UT 2215.03 BOOL  ; Z
V0120_INN 2520.15 BOOL  ; Z
V0120_UT 2220.15 BOOL  ; Z
V0142_INN 2519.01 BOOL  ; Z
V0142_UT 2219.01 BOOL  ; Z
V0143_INN 2519.02 BOOL  ; Z
V0143_UT 2219.02 BOOL  ; Z
V0144_INN 2519.08 BOOL  ; Z
V0144_LINJE_INAKTIV 703.12 BOOL  ; VENTIL STENGT. INGEN AKTIVITET PAA L1.2
V0144_UT 2219.08 BOOL  ; Z
V0145_INN 2519.09 BOOL  ; Z
V0145_UT 2219.09 BOOL  ; Z
V0146_INN 2516.03 BOOL
V0146_UT 2216.03 BOOL
V0147_INN 2516.06 BOOL
V0147_UT 2216.06 BOOL
V0150_INN 2519.06 BOOL  ; Z
V0150_UT 2219.06 BOOL  ; Z
V0151_INN 2519.14 BOOL  ; Z
V0151_UT 2219.14 BOOL  ; Z
V0153_AUTOPAADRAG D20892 UINT
V0153_D D20823 CHANNEL
V0153_D_MEM D25103 CHANNEL
V0153_ER_TEMP D2030 WORD
V0153_HAST_UT D20898 INT
V0153_I D20822 CHANNEL
V0153_I_MEM D25102 CHANNEL
V0153_MAN_AAPNING D2034 WORD
V0153_MAN_AUTO 1001.02 BOOL
V0153_P D20851 CHANNEL
V0153_PRS_TEMP D2032 WORD
V0153_P_MEM D25101 CHANNEL
V0153_REGN1 D20894 REAL
V0153_REGN2 D20896 REAL
V0153_RESET_REG D20850 CHANNEL
V0153_UT D1450 CHANNEL  ; Z
V0154_AUTOPAADRAG D20942 UINT
V0154_D D20803 CHANNEL
V0154_D_MEM D25113 CHANNEL
V0154_ER_TEMP D2130 WORD
V0154_HAST_UT D20948 INT
V0154_I D20902 CHANNEL
V0154_I_MEM D25112 CHANNEL
V0154_MAN_AAPNING D2134 WORD
V0154_MAN_AUTO 1001.03 BOOL
V0154_P D20901 CHANNEL
V0154_PRS_TEMP D2132 WORD
V0154_P_MEM D25111 CHANNEL
V0154_REGN1 D20944 REAL
V0154_REGN2 D20946 REAL
V0154_RESET_REG D20900 CHANNEL
V0154_UT D1452 CHANNEL  ; Z
V0201_INN 2520.01 BOOL  ; Z
V0201_UT 2220.01 BOOL  ; Z
V0204_INN 2520.04 BOOL  ; Z
V0204_INN_FORS_S T0090 BOOL
V0204_LINJE_INAKTIV 705.12 BOOL  ; VENTIL STENGT. INGEN AKTIVITET PAA L2.1
V0204_LINJE_INAKTIV_S C0133 BOOL  ; VENTIL STENGT. INGEN AKTIVITET PAA L2.1
V0204_LINJE_INAKTIV_T C133 CHANNEL  ; VENTIL STENGT. INGEN AKTIVITET PAA L2.1
V0204_STENGER 704.14 BOOL
V0204_UT 2220.04 BOOL  ; Z
V0204_UT_FORS_S T0091 BOOL
V0204_UT_ML_FORS_S T0077 BOOL
V0204_UT_ML_FORS_T 077 NUMBER
V0205_INN 2520.05 BOOL  ; Z
V0205_UT 2220.05 BOOL  ; Z
V0206_INN 2520.12 BOOL  ; Z
V0206_UT 2220.12 BOOL  ; Z
V0207_INN 2520.00 BOOL  ; Z
V0207_UT 2220.00 BOOL  ; Z
V0208_INN 2520.13 BOOL  ; Z
V0208_UT 2220.13 BOOL  ; Z
V0209_INN 2518.02 BOOL  ; Z
V0209_UT 2218.02 BOOL  ; Z
V0210_INN 2522.15 BOOL  ; Z
V0210_UT 2222.15 BOOL  ; Z
V0211_INN 2520.07 BOOL  ; Z
V0211_UT 2220.07 BOOL  ; Z
V0214_INN 2520.10 BOOL  ; Z
V0214_INN_FORS_S T0095 BOOL
V0214_LINJE_INAKTIV_S C0134 BOOL  ; VENTIL STENGT. INGEN AKTIVITET PAA L2.2
V0214_LINJE_INAKTIV_T C134 CHANNEL  ; VENTIL STENGT. INGEN AKTIVITET PAA L2.2
V0214_STENGER 706.14 BOOL
V0214_UT 2220.10 BOOL  ; Z
V0214_UT_FORS_S T0096 BOOL
V0214_UT_ML_FORS_S T0078 BOOL
V0214_UT_ML_FORS_T 078 NUMBER
V0215_INN 2520.11 BOOL  ; Z
V0215_UT 2220.11 BOOL  ; Z
V0217_INN 2518.01 BOOL  ; Z
V0217_UT 2218.01 BOOL  ; Z
V0220_INN 2522.07 BOOL  ; Z
V0220_UT 2222.07 BOOL  ; Z
V0242_INN 2520.02 BOOL  ; Z
V0242_UT 2220.02 BOOL  ; Z
V0243_INN 2520.03 BOOL  ; Z
V0243_UT 2220.03 BOOL  ; Z
V0244_INN 2520.08 BOOL  ; Z
V0244_UT 2220.08 BOOL  ; Z
V0245_INN 2520.09 BOOL  ; Z
V0245_UT 2220.09 BOOL  ; Z
V0246_INN 2516.08 BOOL
V0246_UT 2216.08 BOOL
V0247_INN 2516.09 BOOL
V0247_UT 2216.09 BOOL
V0250_INN 2520.06 BOOL  ; Z
V0250_UT 2220.06 BOOL  ; Z
V0251_INN 2520.14 BOOL  ; Z
V0251_UT 2220.14 BOOL  ; Z
V0253_AUTOPAADRAG D20992 UINT
V0253_D D20923 CHANNEL
V0253_D_MEM D25123 CHANNEL
V0253_ER_TEMP D2230 WORD
V0253_HAST_UT D20998 INT
V0253_I D20922 CHANNEL
V0253_I_MEM D25122 CHANNEL
V0253_MAN_AAPNING D2234 WORD
V0253_MAN_AUTO 1001.04 BOOL
V0253_P D20951 CHANNEL
V0253_PRS_TEMP D2232 WORD
V0253_P_MEM D25121 CHANNEL
V0253_REGN1 D20994 REAL
V0253_REGN2 D20996 REAL
V0253_RESET_REG D20950 CHANNEL
V0253_UT D1454 CHANNEL  ; Z
V0254_AUTOPAADRAG D21042 UINT
V0254_D D21003 CHANNEL
V0254_D_MEM D25133 CHANNEL
V0254_ER_TEMP D2330 WORD
V0254_HAST_UT D21048 INT
V0254_I D21002 CHANNEL
V0254_I_MEM D25132 CHANNEL
V0254_MAN_AAPNING D2334 WORD
V0254_MAN_AUTO 1001.05 BOOL
V0254_P D21001 CHANNEL
V0254_PRS_TEMP D2332 WORD
V0254_P_MEM D25131 CHANNEL
V0254_REGN1 D21044 REAL
V0254_REGN2 D21046 REAL
V0254_RESET_REG D21000 CHANNEL
V0254_UT D1456 CHANNEL  ; Z
V0301_INN 2503.05 BOOL  ; Z
V0301_UT 2203.05 BOOL  ; Z
V0302_INN 2522.03 BOOL  ; Z
V0302_UT 2222.03 BOOL  ; Z
V0303_INN 2522.04 BOOL  ; Z
V0303_UT 2222.04 BOOL  ; Z
V0304_INN 2522.05 BOOL  ; Z
V0304_NEDRE 2223.01 BOOL
V0304_OEVRE 2223.00 BOOL
V0304_UT 2222.05 BOOL  ; Z
V0305_INN 2522.06 BOOL  ; Z
V0305_UT 2222.06 BOOL  ; Z
V0306_INN 2522.08 BOOL  ; Z
V0306_UT 2222.08 BOOL  ; Z
V0307_INN 2521.15 BOOL  ; Z
V0307_UT 2221.15 BOOL  ; Z
V0308_INN 2521.10 BOOL  ; Z
V0308_UT 2221.10 BOOL  ; Z
V0309_INN 2522.02 BOOL  ; Z
V0309_UT 2222.02 BOOL  ; Z
V0310_INN 2521.12 BOOL  ; Z
V0310_NEDRE 2223.07 BOOL
V0310_OEVRE 2223.06 BOOL
V0310_UT 2221.12 BOOL  ; Z
V0312_INN 2516.13 BOOL  ; Z
V0312_UT 2216.13 BOOL  ; Z
V0313_INN 2516.11 BOOL  ; Z
V0313_UT 2216.11 BOOL  ; Z
V0315_INN 2522.12 BOOL  ; Z
V0315_UT 2222.12 BOOL  ; Z
V0319_INN 2515.15 BOOL  ; Z
V0319_UT 2215.15 BOOL  ; Z
V0320_INN 2521.11 BOOL  ; Z
V0320_NEDRE 2223.09 BOOL
V0320_OEVRE 2223.08 BOOL
V0320_UT 2221.11 BOOL  ; Z
V0321_INN 2503.11 BOOL  ; Z
V0321_UT 2203.11 BOOL  ; Z
V0322_INN 2516.10 BOOL  ; Z
V0322_UT 2216.10 BOOL  ; Z
V0328_INN 2521.03 BOOL  ; Z
V0328_UT 2221.03 BOOL  ; Z
V0329_UT 2225.00 BOOL  ; Z
V0330_INN 2521.14 BOOL  ; Z
V0330_NEDRE 2223.11 BOOL
V0330_OEVRE 2223.10 BOOL
V0330_UT 2221.14 BOOL  ; Z
V0332_INN 2517.02 BOOL  ; Z
V0332_UT 2217.02 BOOL  ; Z
V0333_INN 2517.00 BOOL  ; Z
V0333_UT 2217.00 BOOL  ; Z
V0338_INN 2521.04 BOOL  ; Z
V0338_UT 2221.04 BOOL  ; Z
V0339_UT 2225.01 BOOL  ; V0416_OE_UT
V0340_INN 2521.13 BOOL  ; Z
V0340_NEDRE 2223.13 BOOL
V0340_OEVRE 2223.12 BOOL
V0340_UT 2221.13 BOOL  ; Z
V0342_INN 2516.15 BOOL  ; Z
V0342_UT 2216.15 BOOL  ; Z
V0350_INN 2508.00 BOOL  ; Z
V0350_UT 2208.00 BOOL  ; Z
V0351_INN 2508.03 BOOL  ; Z
V0351_UT 2208.03 BOOL  ; Z
V0352_INN 2506.02 BOOL  ; Z
V0352_UT 2206.02 BOOL  ; Z
V0355_INN 2534.02 BOOL
V0355_UT 2234.02 BOOL
V0356_INN 2534.01 BOOL
V0356_UT 2234.01 BOOL
V0357_INN 2534.04 BOOL
V0357_UT 2234.04 BOOL
V0358_INN 2540.01 BOOL
V0358_UT 2240.01 BOOL
V0359_INN 2506.08 BOOL  ; Z
V0359_UT 2206.08 BOOL  ; Z
V0360_INN 2506.14 BOOL  ; Z
V0360_UT 2206.14 BOOL  ; Z
V0362_INN 2522.00 BOOL  ; Z
V0362_UT 2222.00 BOOL  ; Z
V0365_INN 2534.00 BOOL
V0365_UT 2234.00 BOOL
V0366_INN 2534.03 BOOL
V0366_UT 2234.03 BOOL
V0368_INN 2540.02 BOOL
V0368_UT 2240.02 BOOL
V0370_INN 2503.08 BOOL  ; Z
V0370_UT 2203.08 BOOL  ; V0302_OE_UT
V0371_INN 2522.13 BOOL  ; Z
V0371_UT 2222.13 BOOL  ; Z
V0401_INN 2504.07 BOOL  ; Z
V0401_INN_PR2 5129.10 BOOL
V0401_UT 2204.07 BOOL  ; Z
V0401_UT_PR2 5020.10 BOOL
V0402_INN 2505.05 BOOL  ; Z
V0402_NEDRE 2205.07 BOOL
V0402_OEVRE 2205.06 BOOL
V0402_UT 2205.05 BOOL  ; Z
V0403_INN 2553.02 BOOL
V0403_UT 2253.02 BOOL
V0404_INN 2514.03 BOOL  ; Z
V0404_NEDRE 2223.03 BOOL
V0404_OEVRE 2223.02 BOOL
V0404_UT 2214.03 BOOL  ; Z
V0405_INN 2514.04 BOOL  ; Z
V0405_UT 2214.04 BOOL  ; Z
V0406_INN 2504.04 BOOL  ; Z
V0406_NEDRE 2253.01 BOOL
V0406_OEVRE 2253.00 BOOL
V0406_UT 2204.04 BOOL  ; Z
V0407_INN 2521.01 BOOL  ; Z
V0407_UT 2221.01 BOOL  ; Z
V0408_INN 2521.02 BOOL  ; Z
V0408_OEVRE 2229.05 BOOL
V0408_OEVRE_UT 2229.05 BOOL
V0408_OEVRE_UT_PR3 5200.03 BOOL
V0408_UT 2221.02 BOOL  ; Z
V0409_INN 2514.00 BOOL  ; Z
V0409_INN_PR2 5143.01 BOOL
V0409_UT 2214.00 BOOL  ; V0418_UT
V0409_UT_PR2 5024.01 BOOL
V0410_INN 2515.07 BOOL  ; Z
V0410_NEDRE 2223.15 BOOL
V0410_OEVRE 2223.14 BOOL
V0410_UT 2215.07 BOOL  ; Z
V0414_INN 2553.03 BOOL
V0414_UT 2253.03 BOOL
V0415_INN 2504.08 BOOL  ; Z
V0415_UT 2204.08 BOOL  ; Z
V0419_INN 2517.03 BOOL  ; Z
V0419_NEDRE 2217.05 BOOL
V0419_OEVRE 2217.04 BOOL
V0419_UT 2217.03 BOOL  ; Z
V0420_INN 2515.06 BOOL  ; Z
V0420_NEDRE 2224.01 BOOL
V0420_OEVRE 2224.00 BOOL
V0420_UT 2215.06 BOOL  ; Z
V0421_INN 2504.09 BOOL  ; Z
V0421_UT 2204.09 BOOL  ; Z
V0428_INN 2522.11 BOOL  ; Z
V0428_UT 2222.11 BOOL  ; Z
V0429_UT 2225.02 BOOL  ; Z
V0430_INN 2515.09 BOOL  ; Z
V0430_NEDRE 2224.03 BOOL
V0430_OEVRE 2224.02 BOOL
V0430_UT 2215.09 BOOL  ; Z
V0438_INN 2522.09 BOOL  ; Z
V0438_UT 2222.09 BOOL  ; Z
V0439_UT 2225.03 BOOL  ; Z
V0440_INN 2515.08 BOOL  ; Z
V0440_NEDRE 2224.05 BOOL
V0440_OEVRE 2224.04 BOOL
V0440_UT 2215.08 BOOL  ; Z
V0450_INN 2504.12 BOOL  ; Z
V0450_UT 2204.12 BOOL  ; Z
V0459_INN 2521.05 BOOL  ; V0319_N_INN
V0459_UT 2221.05 BOOL  ; V0319_N_UT
V0460_INN 2504.10 BOOL  ; Z
V0460_UT 2204.10 BOOL  ; Z
V0470_INN 2514.13 BOOL  ; Z
V0470_UT 2214.13 BOOL  ; V0516_OEvre
V0471_INN 2521.09 BOOL  ; V0319_OE_INN
V0471_UT 2221.09 BOOL  ; V0319_OE_UT
V0480_INN 2518.12 BOOL  ; Z
V0480_UT 2218.12 BOOL
V0481_INN 2518.04 BOOL  ; Z
V0481_UT 2218.04 BOOL  ; Z
V0482_INN_LUKKET 2518.11 BOOL  ; Z
V0482_INN_OPEN 2515.05 BOOL  ; Z
V0482_TIDSFORINKELSE T0450 BOOL
V0482_UT_LUKKE 2218.11 BOOL  ; Z
V0482_UT_OPNE 2215.05 BOOL  ; Z
V0501_INN 2516.04 BOOL  ; Z
V0501_UT 2216.04 BOOL  ; Z
V0502_INN 2514.06 BOOL  ; Z
V0502_NEDRE 2253.11 BOOL
V0502_OEVRE 2253.12 BOOL
V0502_UT 2214.06 BOOL  ; Z
V0503_INN 2514.07 BOOL  ; Z
V0503_UT 2214.07 BOOL  ; Z
V0504_INN 2514.08 BOOL  ; Z
V0504_NEDRE 2223.05 BOOL
V0504_OEVRE 2223.04 BOOL
V0504_UT 2214.08 BOOL  ; Z
V0505_INN 2514.09 BOOL  ; Z
V0505_UT 2214.09 BOOL  ; Z
V0506_INN 2516.05 BOOL  ; Z
V0506_NEDRE 2253.09 BOOL
V0506_OEVRE 2253.08 BOOL
V0506_UT 2216.05 BOOL  ; Z
V0507_INN 2515.12 BOOL  ; Z
V0507_UT 2215.12 BOOL  ; Z
V0508_INN 2506.05 BOOL  ; Z
V0508_UT 2206.05 BOOL  ; Z
V0509_INN 2514.05 BOOL  ; Z
V0509_UT 2214.05 BOOL  ; V0516_N
V0510_INN 2516.00 BOOL  ; Z
V0510_UT 2216.00 BOOL  ; Z
V0514_INN 2553.10 BOOL
V0514_UT 2253.10 BOOL
V0515_INN 2521.08 BOOL  ; Z
V0515_UT 2221.08 BOOL  ; Z
V0517_UT 2215.00 BOOL
V0519_INN 2504.11 BOOL  ; Z
V0519_NEDRE 2253.06 BOOL
V0519_OEVRE 2253.05 BOOL
V0519_UT 2204.11 BOOL  ; Z
V0520_INN 2515.14 BOOL  ; Z
V0520_UT 2215.14 BOOL  ; Z
V0521_INN 2515.13 BOOL  ; Z
V0521_UT 2215.13 BOOL  ; Z
V0528_INN 2522.14 BOOL  ; Z
V0528_UT 2222.14 BOOL  ; Z
V0529_UT 2225.04 BOOL  ; Z
V0530_INN 2516.02 BOOL  ; Z
V0530_UT 2216.02 BOOL  ; Z
V0538_INN 2522.10 BOOL  ; Z
V0538_UT 2222.10 BOOL  ; Z
V0539_UT 2225.05 BOOL  ; Z
V0540_INN 2516.01 BOOL  ; Z
V0540_UT 2216.01 BOOL  ; Z
V0550_INN 2504.14 BOOL  ; Z
V0550_UT 2204.14 BOOL  ; Z
V0553_INN 2505.02 BOOL  ; Z
V0553_UT 2205.02 BOOL  ; Z
V0554_UT 2214.10 BOOL  ; Z
V0559_INN 2516.07 BOOL  ; Z
V0559_UT 2216.07 BOOL  ; Z
V0560_INN 2505.01 BOOL  ; Z
V0560_UT 2205.01 BOOL  ; Z
V0561_INN 2505.15 BOOL  ; Z
V0561_UT 2205.15 BOOL  ; Z
V0563_INN 2505.00 BOOL  ; Z
V0563_UT 2205.00 BOOL  ; Z
V0564_INN 2505.03 BOOL  ; Z
V0564_UT 2205.03 BOOL  ; Z
V0565_INN 2503.14 BOOL  ; Z
V0565_UT 2203.14 BOOL  ; Z
V0566_UT 2214.12 BOOL  ; Z
V0570_INN 2515.00 BOOL  ; Z
V0570_UT 2215.00 BOOL  ; V0517_UT
V0571_INN 2521.06 BOOL  ; Z
V0571_UT 2221.06 BOOL  ; V0302_N_UT
V0580_INN 2506.11 BOOL  ; Z
V0580_UT 2206.11 BOOL  ; Z
V0581_INN 2503.02 BOOL  ; Z
V0581_UT 2203.02 BOOL  ; Z
V0582_INN_LUKKET 2553.14 BOOL
V0582_INN_OPEN 2553.04 BOOL
V0582_TIDSFORINKELSE T0451 BOOL
V0582_UT_LUKKE 2253.14 BOOL
V0582_UT_OPNE 2253.04 BOOL
V0601_INN 2514.11 BOOL  ; TIL NODE1
V0601_INN_PR2 5129.00 BOOL  ; TIL NODE1
V0601_UT 2214.11 BOOL  ; Z
V0601_UT_PR2 5020.00 BOOL  ; FRA NODE1
V0602_INN 2525.06 BOOL
V0602_UT 2225.06 BOOL
V0604_INN 2525.07 BOOL
V0604_INN_PR2 5129.02 BOOL  ; TIL NODE1
V0604_UT 2225.07 BOOL
V0604_UT_PR2 5020.02 BOOL  ; FRA NODE1
V0605_INN 2525.08 BOOL
V0605_INN_PR2 5129.03 BOOL  ; TIL NODE1
V0605_UT 2225.08 BOOL
V0605_UT_PR2 5020.03 BOOL  ; FRA NODE1
V0640_INN 2525.13 BOOL
V0640_UT 2225.13 BOOL
V0640_UT_N5 2846.00 BOOL
V0641_INN 2525.14 BOOL
V0641_UT 2225.14 BOOL
V0641_UT_N5 2846.01 BOOL
V0642_INN 2525.15 BOOL
V0642_UT 2225.15 BOOL
V0642_UT_N5 2846.02 BOOL
V0643_INN 2526.03 BOOL
V0643_UT 2226.03 BOOL
V0643_UT_N5 2846.03 BOOL
V0644_INN 2526.04 BOOL
V0644_UT 2226.04 BOOL
V0644_UT_N5 2846.04 BOOL
V0651_INN 2525.09 BOOL
V0651_UT 2225.09 BOOL
V0652_INN 2525.10 BOOL
V0652_UT 2225.10 BOOL
V0653_INN 2525.11 BOOL
V0653_INN_PR2 5129.07 BOOL  ; TIL NODE1
V0653_UT 2225.11 BOOL
V0653_UT_PR2 5020.07 BOOL  ; FRA NODE1
V0654_INN 2525.12 BOOL
V0654_INN_PR2 5129.08 BOOL  ; TIL NODE1
V0654_UT 2225.12 BOOL
V0654_UT_PR2 5020.08 BOOL  ; FRA NODE1
V0655_INN 2517.01 BOOL
V0655_UT 2217.01 BOOL
V0920_INN 2533.05 BOOL
V0920_UT 2233.05 BOOL
V0921_INN 2533.04 BOOL
V0921_UT 2233.04 BOOL
V0922_INN 2533.06 BOOL
V0922_UT 2233.06 BOOL
V0923_INN 2533.03 BOOL
V0923_UT 2233.03 BOOL
V1141_INN_PR 5124.00 BOOL  ; TIL NODE1
V1141_MAN_COM_BIT 1151.01 BOOL  ; V1141 AAPNES MANUELT FRA DISPLAY TRAKT UHT
V1141_MAN_COM_BIT_N5 2843.01 BOOL
V1141_UT_PR2 5015.00 BOOL  ; FRA NODE1
V1241_INN_PR 5124.01 BOOL  ; TIL NODE1
V1241_MAN_COM_BIT 1151.02 BOOL  ; V1241 AAPNES MANUELT FRA DISPLAY TRAKT UHT
V1241_MAN_COM_BIT_N5 2843.02 BOOL
V1241_UT_PR2 5015.01 BOOL  ; FRA NODE1
V1242_INN 2531.15 BOOL
V1242_INN_PR 5124.02 BOOL  ; TIL NODE1
V1242_UT 2231.15 BOOL  ; ¨
V1242_UT_PR2 5015.02 BOOL  ; FRA NODE1
V1341_INN_PR 5124.03 BOOL  ; TIL NODE1
V1341_MAN_COM_BIT 1151.03 BOOL  ; V1341 AAPNES MANUELT FRA DISPLAY TRAKT UHT
V1341_MAN_COM_BIT_N5 2843.03 BOOL
V1341_UT_PR2 5015.03 BOOL  ; FRA NODE1
V1441_INN 2532.01 BOOL
V1441_INN_PR 5124.04 BOOL  ; TIL NODE1
V1441_MAN_COM_BIT 1151.04 BOOL  ; V1441 AAPNES MANUELT FRA DISPLAY TRAKT UHT
V1441_MAN_COM_BIT_N5 2843.04 BOOL
V1441_UT 2232.01 BOOL
V1441_UT_PR2 5015.04 BOOL  ; FRA NODE1
V1541_INN 2532.02 BOOL
V1541_INN_PR 5124.05 BOOL  ; TIL NODE1
V1541_MAN_COM_BIT 1151.05 BOOL  ; V1541 AAPNES MANUELT FRA DISPLAY TRAKT UHT
V1541_MAN_COM_BIT_N5 2843.05 BOOL
V1541_UT 2232.02 BOOL
V1541_UT_PR2 5015.05 BOOL  ; FRA NODE1
V1641_INN 2532.03 BOOL
V1641_INN_PR 5124.06 BOOL  ; TIL NODE1
V1641_MAN_COM_BIT 1151.06 BOOL  ; V1641 AAPNES MANUELT FRA DISPLAY TRAKT UHT
V1641_MAN_COM_BIT_N5 2843.06 BOOL
V1641_UT 2232.03 BOOL
V1641_UT_PR2 5015.06 BOOL  ; FRA NODE1
V1700_INN_PR2 5126.00 BOOL  ; TIL NODE1
V1700_UT_PR2 5017.00 BOOL  ; FRA NODE1
V1701_INN_PR2 5126.01 BOOL  ; TIL NODE1
V1701_UT_PR2 5017.01 BOOL  ; FRA NODE1
V1702_INN_PR2 5126.02 BOOL  ; TIL NODE1
V1702_UT_PR2 5017.02 BOOL  ; FRA NODE1
V1703_INN_PR2 5126.03 BOOL  ; TIL NODE1
V1703_UT_PR2 5017.03 BOOL  ; FRA NODE1
V1704_INN_PR2 5126.04 BOOL  ; TIL NODE1
V1704_UT_PR2 5017.04 BOOL  ; FRA NODE1
V1705_INN_PR2 5126.05 BOOL  ; TIL NODE1
V1705_UT_PR2 5017.05 BOOL  ; FRA NODE1
V1706_INN_PR2 5126.06 BOOL  ; TIL NODE1
V1706_UT_PR2 5017.06 BOOL  ; FRA NODE1
V1707_UT_PR2 5017.07 BOOL  ; FRA NODE1
V1741_INN 2532.04 BOOL
V1741_INN_PR 5124.07 BOOL  ; TIL NODE1
V1741_MAN_COM_BIT 1151.07 BOOL  ; V1741 AAPNES MANUELT FRA DISPLAY TRAKT UHT
V1741_MAN_COM_BIT_N5 2843.07 BOOL
V1741_UT 2232.04 BOOL  ; FRA NODE1
V1741_UT_PR2 5015.07 BOOL  ; FRA NODE1
V1841_INN 2532.05 BOOL
V1841_INN_PR 5124.08 BOOL  ; TIL NODE1
V1841_MAN_COM_BIT 1151.08 BOOL  ; V1841 AAPNES MANUELT FRA DISPLAY TRAKT UHT
V1841_MAN_COM_BIT_N5 2843.08 BOOL
V1841_UT 2232.05 BOOL
V1841_UT_PR2 5015.08 BOOL  ; FRA NODE1
V1941_INN 2532.06 BOOL
V1941_INN_PR 5124.09 BOOL  ; TIL NODE1
V1941_MAN_COM_BIT 1151.09 BOOL  ; V1941 AAPNES MANUELT FRA DISPLAY TRAKT UHT
V1941_MAN_COM_BIT_N5 2843.09 BOOL
V1941_UT 2232.06 BOOL  ; FRA NODE1
V1941_UT_PR2 5015.09 BOOL  ; FRA NODE1
V1943_INN 2532.07 BOOL  ; TIL NODE1
V1943_INN_PR 5124.10 BOOL  ; TIL NODE1
V1943_UT 2232.07 BOOL  ; FRA NODE1
V1943_UT_PR2 5015.10 BOOL  ; FRA NODE1
V2001_INN_N5 2827.08 BOOL
V2001_INN_PR2 5128.00 BOOL  ; TIL NODE1
V2001_UT_PR2 5019.00 BOOL  ; FRA NODE1
V2002_INN_N5 2827.09 BOOL
V2002_INN_PR2 5128.02 BOOL  ; TIL NODE1
V2002_UT_PR2 5019.02 BOOL  ; FRA NODE1
V2003_INN_N5 2827.10 BOOL
V2003_INN_PR2 5128.03 BOOL  ; TIL NODE1
V2003_UT_PR2 5019.03 BOOL  ; FRA NODE1
V2004_INN_N5 2827.11 BOOL
V2004_INN_PR2 5128.04 BOOL  ; TIL NODE1
V2004_UT_PR2 5019.04 BOOL  ; FRA NODE1
V204_INNT_FORS_T 090 NUMBER
V204_UT_FORS_T 091 NUMBER
V2101_INN 2534.05 BOOL
V2101_UT 2234.05 BOOL
V2104_INN 2534.06 BOOL
V2104_UT 2234.06 BOOL
V2106_INN 2534.07 BOOL
V2106_UT 2234.07 BOOL
V2107_INN 2534.08 BOOL
V2107_UT 2234.08 BOOL  ; ¨
V2108_INN 2534.09 BOOL
V2108_UT 2234.09 BOOL
V2111_INN 2534.10 BOOL
V2111_UT 2234.10 BOOL
V2112_INN 2534.11 BOOL
V2112_UT 2234.11 BOOL
V2113_INN 2534.12 BOOL  ; ,
V2113_UT 2234.12 BOOL
V2114_INN 2534.13 BOOL
V2114_UT 2234.13 BOOL
V2119_ADV BRA_PID_ADV1
V2119_D D3194 INT  ; 0_1000
V2119_I D3193 INT  ; 0_1000
V2119_INN 2534.14 BOOL
V2119_MAN_AUTO 1002.00 BOOL  ; MAN=1
V2119_MAN_PRS D3196 UINT  ; 0-1000
V2119_OPPSKALER OPPSKALERING
V2119_P D3192 INT  ; 0_1000
V2119_PAADRAG D3190 INT  ; 0_1000
V2119_PAADRAG_HJ D3191 INT  ; 0_1000
V2119_PRS_TRYKK D3188 INT  ; 0_7,00 BAR
V2119_UT 2234.14 BOOL
V2120_INN 2534.15 BOOL
V2120_UT 2234.15 BOOL
V2121_INN 2535.00 BOOL
V2121_UT 2235.00 BOOL
V2122_INN 2535.01 BOOL
V2122_UT 2235.01 BOOL
V2132_UT 2205.09 BOOL
V2133_INN 2535.02 BOOL
V2133_UT 2235.02 BOOL
V2140_INN 2535.03 BOOL
V2140_UT 2235.03 BOOL
V2141_INN 2535.04 BOOL
V2141_UT 2235.04 BOOL
V2142_INN 2535.05 BOOL
V2142_UT 2235.05 BOOL
V2144_INN 2535.06 BOOL
V2144_LINJE_INAKTIV 707.12 BOOL  ; VENTIL STENGT. INGEN AKTIVITET PAA L2.2
V2144_UT 2235.06 BOOL
V2145_INN 2535.07 BOOL
V2145_UT 2235.07 BOOL
V2146_INN 2535.08 BOOL
V2146_UT 2235.08 BOOL
V214_INN_FORS_T 095 NUMBER
V214_UT_FORS_T 096 NUMBER
V2150_INN 2535.09 BOOL
V2150_UT 2235.09 BOOL
V2154_INN 2535.10 BOOL
V2154_UT 2235.10 BOOL
V2161 BRA_PID
V2161_AAPNING_0_1000 D1412 UINT  ; 0-1000
V2161_AKTUELT_PRS D3126 WORD  ; AKTUELL PRS VED OPP- ELLER NEDTRAPPING
V2161_AKT_PRS_S T0481 BOOL
V2161_AKT_PRS_T 0481 NUMBER
V2161_AKT_UT_PRS_S T0482 BOOL
V2161_AKT_UT_PRS_T 0482 NUMBER
V2161_C23_AKT_UT_PRS D3152 WORD
V2161_C23_DIF_VSP_ASP D3150 WORD  ; DIFF MELLOM VALGT PRS OG AKTUELL PRS
V2161_C23_FORRIGE_AKTUELLE_PRS D3148 WORD  ; AKTUELL PRS VED OPP- ELLER NEDTRAPPING
V2161_D D22053 CHANNEL
V2161_DIFF_PRS_HJ1 D3142 WORD  ; HJ  DIFFERANSE MELLOM AKTUELT SETP. OG VALGT SETP
V2161_DIFF_PRS_HJ2 D3144 WORD  ; HJ  DIFFERANSE MELLOM AKTUELT SETP. OG VALGT SETP
V2161_DIFF_PRS_VALGT_ER D3140 WORD  ; DIFFERANSE MELLOM AKTUELT SETP. OG VALGT SETP
V2161_FORRIGE_AKTUELLE_PRS D3138 WORD  ; AKTUELL PRS VED OPP- ELLER NEDTRAPPING
V2161_HJ_PRS_VALGT D3134 WORD  ; D3130 + 3 GRADER
V2161_I D22052 CHANNEL
V2161_MAN_AUTO 1001.08 BOOL
V2161_NY_DIFF D3146 WORD  ; ENDRE SETPUNKT MED 0.5 AV DIFF
V2161_OPPSKALER OPPSKALERING
V2161_P D22051 CHANNEL
V2161_PRS_FORIG_VALGTE_PRS D3132 WORD
V2161_PRS_MAN D3128 WORD
V2161_PRS_OEKES 4800.02 BOOL
V2161_PRS_SENKES 4800.01 BOOL
V2161_PRS_VALGT D3130 WORD
V2161_VALGT_PRS_MIN 4800.00 BOOL
V2161_VALGT_PRS_MIN_S T0480 BOOL
V2161_VALGT_PRS_MIN_T 0480 NUMBER
V2174_INN 2535.11 BOOL
V2174_UT 2235.11 BOOL
V2201_INN 2535.12 BOOL
V2201_S T0836 BOOL  ; FORSINKER FRAFALL
V2201_T 0836 NUMBER  ; FORSINKER FRAFALL
V2201_UT 2235.12 BOOL
V2204_INN 2535.13 BOOL
V2204_UT 2235.13 BOOL
V2206_INN 2535.14 BOOL
V2206_UT 2235.14 BOOL
V2207_INN 2535.15 BOOL
V2207_UT 2235.15 BOOL
V2208_INN 2536.00 BOOL
V2208_UT 2236.00 BOOL
V2211_INN 2536.01 BOOL
V2211_UT 2236.01 BOOL
V2212_INN 2536.02 BOOL
V2212_UT 2236.02 BOOL
V2213_INN 2536.03 BOOL
V2213_UT 2236.03 BOOL
V2214_INN 2536.04 BOOL
V2214_UT 2236.04 BOOL
V2216_INN 2536.05 BOOL
V2216_UT 2236.05 BOOL
V2217_INN 2536.06 BOOL
V2217_UT 2236.06 BOOL
V2218_INN 2536.07 BOOL
V2218_UT 2236.07 BOOL
V2219_ADV BRA_PID_ADV1
V2219_D D3294 UINT  ; 0_1000
V2219_I D3293 UINT  ; 0_1000
V2219_INN 2536.08 BOOL
V2219_MAN_AUTO 1001.15 BOOL  ; MAN=1
V2219_MAN_PRS D3296 UINT  ; 0-1000
V2219_OPPSKALER OPPSKALERING
V2219_P D3292 UINT  ; 0_1000
V2219_PAADRAG D3290 UINT  ; 0_1000
V2219_PRS_TRYKK D3288 UINT  ; 0_7,00 BAR
V2219_UT 2236.08 BOOL
V2220_INN 2536.09 BOOL
V2220_UT 2236.09 BOOL
V2221_INN 2536.10 BOOL
V2221_UT 2236.10 BOOL
V2222_INN 2536.11 BOOL
V2222_UT 2236.11 BOOL
V2223_INN 2536.12 BOOL
V2223_S T0837 BOOL  ; FORSINKET FRAFALL
V2223_T 0837 NUMBER  ; FORSINKET FRAFALL
V2223_UT 2236.12 BOOL
V2224_INN 2536.13 BOOL
V2224_S T0838 BOOL  ; FORSINKET FRAFALL
V2224_T 0838 NUMBER  ; FORSINKET FRAFALL
V2224_UT 2236.13 BOOL
V2225_INN 2536.14 BOOL
V2225_UT 2236.14 BOOL
V2240_INN 2536.15 BOOL
V2240_UT 2236.15 BOOL
V2241_INN 2537.00 BOOL
V2241_UT 2237.00 BOOL
V2242_INN 2537.01 BOOL
V2242_UT 2237.01 BOOL
V2244_INN 2537.02 BOOL
V2244_UT 2237.02 BOOL
V2246_INN 2537.03 BOOL
V2246_UT 2237.03 BOOL
V2247_INN 2537.04 BOOL
V2247_UT 2237.04 BOOL
V2248_INN 2537.05 BOOL
V2248_UT 2237.05 BOOL
V2249_INN 2537.06 BOOL
V2249_UT 2237.06 BOOL
V2250_INN 2537.07 BOOL
V2250_UT 2237.07 BOOL
V2251_INN 2540.05 BOOL
V2251_UT 2240.05 BOOL
V2252 BRA_PID
V2252_D D23013 CHANNEL
V2252_I D23012 CHANNEL
V2252_MAN_AUTO 1001.10 BOOL
V2252_MAN_PRS D3226 WORD  ; 0-1000
V2252_OPPSKALER OPPSKALERING
V2252_P D23011 CHANNEL
V2252_PAADRAG D1414 UINT
V2252_PRS D3224 WORD  ; 0-1000
V2254_INN 2537.08 BOOL
V2254_UT 2237.08 BOOL
V2255_INN 2537.09 BOOL
V2255_UT 2237.09 BOOL
V2256_INN 2537.10 BOOL
V2256_UT 2237.10 BOOL
V2257_INN 2537.11 BOOL
V2257_UT 2237.11 BOOL
V2261 BRA_PID
V2261_AKTUELT_PRS D3236 WORD  ; '
V2261_C24_AKT_UT_PRS D3272 WORD
V2261_C24_DIF_VALGT_AKT_PRS D3282 WORD
V2261_C24_DIF_VSP_ASP D3270 WORD  ; DIFF MELLOM VALGT PRS OG AKTUELL PRS
V2261_C24_FORRIGE_AKTS D3280 WORD
V2261_C24_FORRIGE_AKTUELLE_PRS D3268 WORD  ; AKTUELL PRS VED OPP- ELLER NEDTRAPPING
V2261_D D23033 CHANNEL
V2261_DIFF_PRS_HJ1 D3262 WORD  ; HJ  DIFFERANSE MELLOM AKTUELT SETP. OG VALGT SETP
V2261_DIFF_PRS_HJ2 D3264 WORD  ; HJ  DIFFERANSE MELLOM AKTUELT SETP. OG VALGT SETP
V2261_DIFF_PRS_VALGT_ER D3260 WORD  ; DIFFERANSE MELLOM AKTUELT SETP. OG VALGT SETP
V2261_ER_C24_LES_TIL_F0RIGE_AKTS D3286 WORD
V2261_ER_LES_TIL_F0RIGE_AKTS D3278 WORD
V2261_FORRIGE_AKTUELLE_PRS D3258 WORD  ; AKTUELL PRS VED OPP- ELLER NEDTRAPPING
V2261_HJ_PRS_VALGT D3254 WORD  ; D3250 + 3 GRADER
V2261_I D23032 CHANNEL
V2261_MAN_AUTO 1001.12 BOOL
V2261_MAN_PRS D3238 WORD  ; 0-1000
V2261_NY_DIFF D3266 WORD  ; ENDRE SETPUNKT MED 0.5 AV DIFF
V2261_OK_PRO_LES_TIL_F0RIGE_AKTS 4810.04 BOOL  ; OPROD
V2261_OK_VASK_LES_TIL_F0RIGE_AKTS 4810.05 BOOL
V2261_OPPSKALER OPPSKALERING
V2261_P D23031 CHANNEL
V2261_PAADRAG D1416 UINT  ; 0-1000
V2261_PRS_C24_LES_TIL_F0RIGE_AKTS D3284 WORD
V2261_PRS_FORIG_VALGTE_PRS D3252 WORD
V2261_PRS_LES_TIL_F0RIGE_AKTS D3276 WORD
V2261_PRS_MAN D3238 WORD
V2261_PRS_OEKES 4810.02 BOOL
V2261_PRS_SENKES 4810.01 BOOL
V2261_PRS_VALGT D3250 WORD
V2261_PRS_VALGT_4C D3274 WORD  ; VALGT PRS + 4 GRADER C
V2261_VALGT_PRS_MIN 4810.00 BOOL
V2261_VALGT_PRS_MIN_S T0802 BOOL  ; V2261_SETPUNKT=MIN
V2261_VALGT_PRS_MIN_T 0802 NUMBER  ; V2261_SETPUNKT=MIN
V2274_INN 2537.12 BOOL
V2274_UT 2237.12 BOOL
V2280_SEP22 2217.08 BOOL  ; TRYKK UNDER VASK
V2281_SEP22 2217.07 BOOL  ; VASKETRYKK
V2282_SEP22 2217.06 BOOL  ; TRYKK SURT PODUKT
V2302_INN 2537.14 BOOL
V2302_UT 2237.14 BOOL
V2303_INN 2537.15 BOOL
V2303_UT 2237.15 BOOL
V2304_INN 2541.00 BOOL
V2304_N 2240.11 BOOL
V2304_OE 2240.10 BOOL
V2304_UT 2241.00 BOOL
V2305_INN 2538.01 BOOL
V2305_UT 2238.01 BOOL
V2306_INN 2538.02 BOOL
V2306_UT 2238.02 BOOL
V2307_INN 2541.01 BOOL
V2307_UT 2241.01 BOOL
V2308_INN 2538.03 BOOL
V2308_N 2240.13 BOOL
V2308_OE 2240.12 BOOL
V2308_UT 2238.03 BOOL
V2309_INN 2537.13 BOOL
V2309_UT 2237.13 BOOL
V2310_INN 2532.12 BOOL
V2310_UT 2232.12 BOOL
V2312_MAN 4822.07 BOOL
V2312_OPPSKALER OPPSKALERING
V2312_PAADRAG D1426 UINT
V2312_PID BRA_PID
V2312_PRS_AUTO D3804 INT
V2312_PRS_MAN D3806 INT
V2313_INN 2538.04 BOOL
V2313_UT 2238.04 BOOL
V2314_INN 2538.05 BOOL
V2314_UT 2238.05 BOOL
V2316_INN 2539.10 BOOL
V2316_UT 2239.10 BOOL
V2319_INN 2538.06 BOOL
V2319_UT 2238.06 BOOL
V2320_INN 2538.07 BOOL
V2320_UT 2238.07 BOOL
V2321_INN 2538.08 BOOL
V2321_UT 2238.08 BOOL
V2322_INN 2539.07 BOOL
V2322_UT 2239.07 BOOL
V2323_INN 2532.11 BOOL
V2323_UT 2232.11 BOOL
V2324_INN 2532.13 BOOL
V2324_UT 2232.13 BOOL
V2325_INN 2532.14 BOOL
V2325_UT 2232.14 BOOL
V2326_INN 2538.09 BOOL
V2326_UT 2238.09 BOOL
V2327_INN 2540.04 BOOL
V2327_UT 2240.04 BOOL
V2328_INN 2533.02 BOOL
V2328_UT 2233.02 BOOL  ; TILKOBLET N3
V2330_INN 2533.01 BOOL
V2330_UT 2233.01 BOOL
V2340_INN 2538.10 BOOL
V2340_UT 2238.10 BOOL
V2341_INN 2538.11 BOOL
V2341_UT 2238.11 BOOL
V2342_INN 2538.12 BOOL
V2342_UT 2238.12 BOOL
V2343_INN 2538.13 BOOL
V2343_UT 2238.13 BOOL
V2345_INN 2538.14 BOOL
V2345_UT 2238.14 BOOL
V2346_INN 2532.15 BOOL
V2346_UT 2232.15 BOOL
V2347_INN 2533.00 BOOL
V2347_UT 2233.00 BOOL
V2350_INN 2538.15 BOOL
V2350_STYRESIGN_FRA_V2309 4821.03 BOOL  ; ¨
V2350_UT 2238.15 BOOL
V2351_INN 2539.00 BOOL
V2351_UT 2239.00 BOOL
V2352_INN 2539.01 BOOL
V2352_UT 2239.01 BOOL
V2353_MAN 4826.10 BOOL
V2353_MAN_SETP D3884 INT
V2353_OPPSKALER OPPSKALERING
V2353_PAADRAG D1428 UINT
V2353_REG_SETP D3882 INT
V2354_MAN 4826.11 BOOL
V2354_MAN_SETP D3885 INT
V2354_OPPSKALER OPPSKALERING
V2354_PAADRAG D1430 UINT
V2354_PRS_AUTO D3314 INT
V2354_REG BRA_PID_INV
V2354_REG_SETP D3883 INT  ; ,
V2361 BRA_PID
V2361_AKTUELT_PRS D3346 WORD  ; '
V2361_C24_FORRIGE_AKTS D3390 WORD
V2361_C25_AKT_UT_PRS D3382 WORD
V2361_C25_DIF_VALGT_AKT_PRS D3392 WORD
V2361_C25_DIF_VSP_ASP D3280 WORD  ; DIFF MELLOM VALGT PRS OG AKTUELL PRS
V2361_C25_FORRIGE_AKTUELLE_PRS D3378 WORD  ; AKTUELL PRS VED OPP- ELLER NEDTRAPPING
V2361_D D23053 CHANNEL
V2361_DIFF_PRS_HJ1 D3372 WORD  ; HJ  DIFFERANSE MELLOM AKTUELT SETP. OG VALGT SETP
V2361_DIFF_PRS_HJ2 D3374 WORD  ; HJ  DIFFERANSE MELLOM AKTUELT SETP. OG VALGT SETP
V2361_DIFF_PRS_VALGT_ER D3370 WORD  ; DIFFERANSE MELLOM AKTUELT SETP. OG VALGT SETP
V2361_ER_C25_LES_TIL_F0RIGE_AKTS D3396 WORD
V2361_ER__LES_0_VALGT_PRS D3388 WORD
V2361_FORRIGE_AKTUELLE_PRS D3368 WORD  ; AKTUELL PRS VED OPP- ELLER NEDTRAPPING
V2361_FORRIGE_ER_VERDI D3398 WORD
V2361_HJ_PRS_VALGT D3364 WORD  ; D3250 + 3 GRADER
V2361_I D23052 CHANNEL
V2361_IKKE_PROD 4820.05 BOOL
V2361_MAN_AUTO 1001.14 BOOL  ; MAN=1
V2361_MAN_PRS D3348 WORD  ; 0-1000
V2361_NY_DIFF D3376 WORD  ; ENDRE SETPUNKT MED 0.5 AV DIFF
V2361_OPPSKALER OPPSKALERING
V2361_P D23051 CHANNEL
V2361_PAADRAG D1418 UINT  ; 0-1000
V2361_PROD_ELLER_VASK 4820.06 BOOL
V2361_PRS_0_STILL_S T0885 BOOL
V2361_PRS_0_STILL_T 885 CHANNEL  ; ,
V2361_PRS_C25_LES_TIL_F0RIGE_AKTS D3394 WORD
V2361_PRS_ER_0 4820.03 BOOL
V2361_PRS_FORIG_VALGTE_PRS D3362 WORD
V2361_PRS_LES_0_VALGT_PRS D3386 WORD
V2361_PRS_OEKES 4820.02 BOOL
V2361_PRS_SENKES 4820.01 BOOL
V2361_PRS_TRINNTID D3400 UINT
V2361_PRS_TRINNTID_S T0886 BOOL
V2361_PRS_TRINNTID_T 0886 NUMBER
V2361_PRS_VALGT D3360 WORD  ; ¨
V2361_PRS_VALGT_4C D3384 WORD  ; VALGT PRS + 4 GRADER C
V2361_TID_LES_FAS 4820.04 BOOL
V2361_VALGT_PRS_MIN 4820.00 BOOL
V2363_INN 2538.00 BOOL
V2363_INN_TID_S T0844 BOOL  ; TID V2363 SKAL VAERE AKTIV ETTER AT B2360>0
V2363_UT 2238.00 BOOL
V2401_INN 2539.02 BOOL
V2401_UT 2239.02 BOOL
V2402_INN 2539.03 BOOL
V2402_UT 2239.03 BOOL
V2403_INN 2539.04 BOOL
V2403_UT 2239.04 BOOL
V2406_INN 2539.05 BOOL
V2406_UT 2239.05 BOOL
V2410_INN 2539.06 BOOL
V2410_N 2240.07 BOOL
V2410_OE 2240.06 BOOL  ; '
V2410_UT 2239.06 BOOL
V2412_INN 2539.08 BOOL
V2412_UT 2239.08 BOOL
V2420_INN 2539.09 BOOL
V2420_N 2240.09 BOOL
V2420_OE 2240.08 BOOL
V2420_UT 2239.09 BOOL
V2422_INN 2539.11 BOOL
V2422_UT 2239.11 BOOL
V2429_INN 2540.03 BOOL
V2429_UT 2240.03 BOOL
V2603_INN 2524.14 BOOL  ; MOTTAK OEKOMELK
V2603_INN_PR1 5116.15 BOOL  ; FRA PROFIBUS
V2603_SETELOEFT 2226.06 BOOL
V2603_UT 2224.14 BOOL  ; MOTTAK OEKOMELK
V2603_UT_PR1 5009.15 BOOL  ; TIL PROFIBUS
V2604_INN 2524.15 BOOL  ; MOTTAK OEKOMELK
V2604_UT 2224.15 BOOL  ; MOTTAK OEKOMELK
V2710_INN 2539.12 BOOL
V2710_UT 2239.12 BOOL
V2711_INN 2539.13 BOOL
V2711_UT 2239.13 BOOL
V2712_INN 2539.14 BOOL
V2712_UT 2239.14 BOOL
V3041_UT_N5 2863.08 BOOL
V3335_INN 2550.13 BOOL  ; Z
V3336_INN 2550.14 BOOL  ; Z
V3365_INN 2551.09 BOOL  ; Z
V3366_INN 2551.10 BOOL  ; Z
V3552_INN 2553.15 BOOL  ; Z
V3555_INN 2554.07 BOOL  ; Z
V3610_INN 2531.07 BOOL
V3610_UT 2231.07 BOOL
V3620_INN 2531.08 BOOL
V3620_UT 2231.08 BOOL
V3630_INN 2531.09 BOOL
V3630_UT 2231.09 BOOL
V3640_INN 2531.10 BOOL
V3640_UT 2231.10 BOOL
V3641_INN 2531.04 BOOL
V3641_MAN_COM_BIT 1151.10 BOOL
V3641_MAN_COM_BIT_B 1151.13 BOOL
V3641_MAN_COM_BIT_N5 2843.10 BOOL
V3641_UT 2231.04 BOOL
V3642_INN 2531.05 BOOL
V3642_UT 2231.05 BOOL
V3710_INN 2531.00 BOOL
V3710_UT 2231.00 BOOL
V3720_INN 2531.01 BOOL
V3720_UT 2231.01 BOOL
V3730_INN 2531.02 BOOL
V3730_UT 2231.02 BOOL
V3740_INN 2531.03 BOOL
V3740_UT 2231.03 BOOL
V3741_INN 2531.06 BOOL
V3741_MAN_COM_BIT 1151.11 BOOL
V3741_MAN_COM_BIT_B 1151.14 BOOL
V3741_MAN_COM_BIT_N5 2843.11 BOOL
V3741_UT 2231.06 BOOL
V3742_INN 2531.11 BOOL
V3742_UT 2231.11 BOOL
V3743_INN 2531.12 BOOL
V3743_UT 2231.12 BOOL
V4001_INN 2550.00 BOOL
V4001_UT 2250.00 BOOL
V4002_INN 2550.01 BOOL
V4002_UT 2250.01 BOOL
V4003_INN 2550.02 BOOL
V4003_UT 2250.02 BOOL
V4004_INN 2550.03 BOOL
V4004_UT 2250.03 BOOL
V4005_INN 2550.04 BOOL
V4005_UT 2250.04 BOOL
V4010_INN 2550.05 BOOL
V4010_UT 2250.05 BOOL
V4011_INN 2550.06 BOOL
V4011_UT 2250.06 BOOL
V4012_INN 2550.07 BOOL
V4012_UT 2250.07 BOOL
V4013_INN 2550.08 BOOL
V4013_UT 2250.08 BOOL
V4014_INN 2550.09 BOOL
V4014_UT 2250.09 BOOL
V4015_INN 2550.10 BOOL
V4015_UT 2250.10 BOOL
V4016_INN 2550.11 BOOL
V4016_UT 2250.11 BOOL
V4020_INN 2550.12 BOOL
V4020_UT 2250.12 BOOL
V4060_INN 2550.13 BOOL
V4060_UT 2250.13 BOOL
V4061_INN 2550.14 BOOL
V4061_UT 2250.14 BOOL
V4070_AUTO 1055.10 BOOL
V4070_INN 2550.15 BOOL
V4070_MAN 1005.10 BOOL
V4070_UT 2250.15 BOOL
V4101_INN 2551.00 BOOL
V4101_UT 2251.00 BOOL
V4102_INN 2551.01 BOOL
V4102_UT 2251.01 BOOL
V4103_INN 2551.02 BOOL
V4103_UT 2251.02 BOOL
V4104_INN 2551.03 BOOL
V4104_UT 2251.03 BOOL
V4105_INN 2551.04 BOOL
V4105_UT 2251.04 BOOL
V4110_INN 2551.05 BOOL
V4110_UT 2251.05 BOOL
V4111_INN 2551.06 BOOL  ; CV4401
V4111_UT 2251.06 BOOL
V4120_INN 2551.07 BOOL
V4120_UT 2251.07 BOOL
V4160_INN 2551.08 BOOL
V4160_UT 2251.08 BOOL
V4161_INN 2551.09 BOOL
V4161_UT 2251.09 BOOL
V4170_AUTO 1055.11 BOOL
V4170_INN 2551.10 BOOL
V4170_MAN 1005.11 BOOL
V4170_UT 2251.10 BOOL
V4201_INN 2529.00 BOOL
V4201_INN_PR3 5301.05 BOOL
V4201_UT 2229.00 BOOL
V4201_UT_PR3 5201.05 BOOL
V4202_AKTIV_HJ1 960.06 BOOL
V4202_AKTIV__ALARM_UHT_PR2 5010.05 BOOL  ; FLASH UHT                   V4202  BUNNVENTIL TRAKT UHT TIL DYREFOE ER AKTIVERT. OVER MAX TID
V4202_AKTIV__LAMPE_LAB_PR2 5010.04 BOOL  ; LAMPE VED TRAKT LAB:                    V4202  BUNNVENTIL TRAKT UHT TIL DYREFOE ER AKTIVERT.
V4202_HJ2 960.13 BOOL
V4202_INN 2529.01 BOOL
V4202_INN_PR3 5301.06 BOOL
V4202_MAN_COM_BIT 1150.03 BOOL  ; BUNNVENTIL TRAKT AAPNES MANUELT
V4202_UT 2229.01 BOOL
V4202_UT_PR3 5201.06 BOOL
V4205_INN 2529.02 BOOL
V4205_INN_PR3 5301.07 BOOL
V4205_UT 2229.02 BOOL
V4205_UT_PR3 5201.07 BOOL
V4210_INN 2529.03 BOOL
V4210_INN_PR3 5300.01 BOOL
V4210_UT 2229.03 BOOL
V4210_UT_PR3 5200.01 BOOL
V4211_INN 2529.04 BOOL
V4211_INN_PR3 5300.02 BOOL
V4211_UT 2229.04 BOOL
V4211_UT_PR3 5200.02 BOOL
V4212_INN 2529.05 BOOL
V4212_INN_PR3 5300.03 BOOL
V4212_UT 2229.05 BOOL  ; V0408_OEVRE
V4212_UT_PR3 5200.03 BOOL  ; V0408_OEvre
V4213_INN 2529.06 BOOL
V4213_INN_PR3 5300.04 BOOL
V4213_UT 2229.06 BOOL
V4213_UT_PR3 5200.04 BOOL
V4214_INN 2529.07 BOOL
V4214_INN_PR3 5300.05 BOOL
V4214_UT 2229.07 BOOL  ; V0408_NEDRE
V4214_UT_HJ1 945.03 BOOL
V4214_UT_OFFT_S T0137 BOOL
V4214_UT_OFFT_T 0137 NUMBER
V4214_UT_PR3 5200.05 BOOL  ; V0408_Nedre
V4215_INN 2529.08 BOOL
V4215_INN_PR3 5300.06 BOOL
V4215_UT 2229.08 BOOL
V4215_UT_PR3 5200.06 BOOL
V4218_INN 2529.09 BOOL  ; V0408_INN
V4218_INN_PR3 5300.14 BOOL  ; V0408_INN
V4218_UT 2229.09 BOOL  ; V0408
V4218_UT_OFFT_S T0139 BOOL
V4218_UT_OFFT_T 0139 NUMBER
V4218_UT_ONT_S T0138 BOOL
V4218_UT_ONT_T 0138 NUMBER
V4218_UT_PR3 5200.14 BOOL  ; V0408
V4219_INN 2529.10 BOOL
V4219_INN_PR3 5300.07 BOOL
V4219_UT 2229.10 BOOL
V4219_UT_ONT_S T0140 BOOL
V4219_UT_ONT_T 0140 NUMBER
V4219_UT_PR3 5200.07 BOOL
V4220_INN 2529.11 BOOL
V4220_INN_PR3 5300.08 BOOL
V4220_UT 2229.11 BOOL
V4220_UT_PR3 5200.08 BOOL
V4221_INN 2529.12 BOOL
V4221_INN_PR3 5300.09 BOOL
V4221_UT 2229.12 BOOL
V4221_UT_PR3 5200.09 BOOL
V4222_INN 2529.13 BOOL
V4222_INN_PR3 5300.10 BOOL
V4222_UT 2229.13 BOOL
V4222_UT_PR3 5200.10 BOOL
V4223_INN 2529.14 BOOL
V4223_INN_PR3 5300.11 BOOL
V4223_UT 2229.14 BOOL
V4223_UT_PR3 5200.11 BOOL
V4224_INN 2529.15 BOOL
V4224_INN_PR3 5300.12 BOOL
V4224_UT 2229.15 BOOL
V4224_UT_HJ1 945.04 BOOL
V4224_UT_OFFT_S T0141 BOOL
V4224_UT_OFFT_T 0141 NUMBER
V4224_UT_PR3 5200.12 BOOL
V4225_INN 2530.00 BOOL
V4225_INN_PR3 5300.13 BOOL
V4225_UT 2230.00 BOOL
V4225_UT_PR3 5200.13 BOOL
V4228_INN 2530.01 BOOL
V4228_INN_PR3 5300.15 BOOL
V4228_UT 2230.01 BOOL
V4228_UT_OFFT_S T0143 BOOL
V4228_UT_OFFT_T 0143 NUMBER
V4228_UT_ONT_S T0142 BOOL
V4228_UT_ONT_T 0142 NUMBER
V4228_UT_PR3 5200.15 BOOL
V4230_INN 2530.02 BOOL
V4230_INN_PR3 5301.00 BOOL
V4230_UT 2230.02 BOOL
V4230_UT_PR3 5201.00 BOOL
V4231_INN 2530.03 BOOL
V4231_INN_PR3 5301.01 BOOL
V4231_UT 2230.03 BOOL
V4231_UT_PR3 5201.01 BOOL
V4232_INN 2530.04 BOOL
V4232_INN_PR3 5301.02 BOOL
V4232_UT 2230.04 BOOL
V4232_UT_PR3 5201.02 BOOL
V4233_INN 2530.05 BOOL
V4233_INN_PR3 5301.03 BOOL
V4233_UT 2230.05 BOOL
V4233_UT_PR3 5201.03 BOOL
V4234_INN 2530.06 BOOL
V4234_INN_PR3 5301.04 BOOL
V4234_UT 2230.06 BOOL
V4234_UT_HJ1 945.05 BOOL
V4234_UT_OFFT_S T0144 BOOL
V4234_UT_OFFT_T 0144 NUMBER
V4234_UT_PR3 5201.04 BOOL
V4238_INN 2530.07 BOOL
V4238_INN_PR3 5301.14 BOOL
V4238_UT 2230.07 BOOL
V4238_UT_OFFT_S T0146 BOOL
V4238_UT_OFFT_T 0146 NUMBER
V4238_UT_ONT_S T0145 BOOL
V4238_UT_ONT_T 0145 NUMBER
V4238_UT_PR3 5201.14 BOOL
V4240_INN 2530.08 BOOL
V4240_INN_PR3 5301.08 BOOL
V4240_UT 2230.08 BOOL
V4240_UT_PR3 5201.08 BOOL
V4241_INN 2530.09 BOOL
V4241_INN_PR3 5301.09 BOOL
V4241_UT 2230.09 BOOL
V4241_UT_PR3 5201.09 BOOL
V4242_INN 2530.10 BOOL
V4242_INN_PR3 5301.10 BOOL
V4242_UT 2230.10 BOOL
V4242_UT_PR3 5201.10 BOOL
V4243_INN 2530.11 BOOL
V4243_INN_PR3 5301.11 BOOL
V4243_UT 2230.11 BOOL
V4243_UT_PR3 5201.11 BOOL
V4244_INN 2530.12 BOOL
V4244_INN_PR3 5301.12 BOOL
V4244_UT 2230.12 BOOL
V4244_UT_HJ1 945.06 BOOL
V4244_UT_OFFT_S T0147 BOOL
V4244_UT_OFFT_T 0147 NUMBER
V4244_UT_PR3 5201.12 BOOL
V4245_INN 2530.13 BOOL
V4245_INN_PR3 5301.13 BOOL
V4245_UT 2230.13 BOOL
V4245_UT_PR3 5201.13 BOOL
V4248_INN 2530.14 BOOL
V4248_INN_PR3 5301.15 BOOL
V4248_UT 2230.14 BOOL
V4248_UT_OFFT_S T0149 BOOL
V4248_UT_OFFT_T 0149 NUMBER
V4248_UT_ONT_S T0148 BOOL
V4248_UT_ONT_T 0148 NUMBER
V4248_UT_PR3 5201.15 BOOL
V4249_INN 2530.15 BOOL
V4249_INN_PR3 5300.00 BOOL
V4249_UT 2230.15 BOOL
V4249_UT_ONT_S T0157 BOOL
V4249_UT_ONT_T 0157 NUMBER
V4249_UT_PR3 5200.00 BOOL  ; FRA NODE3
V4250_INN 2532.08 BOOL
V4250_INN_PR 5124.12 BOOL  ; TIL NODE1
V4250_UT 2232.08 BOOL
V4250_UT_N5 2847.11 BOOL
V4250_UT_PR2 5015.12 BOOL  ; FRA NODE1
V4251_INN 2532.09 BOOL
V4251_INN_PR 5124.13 BOOL  ; TIL NODE1
V4251_UT 2232.09 BOOL
V4251_UT_N5 2847.12 BOOL
V4251_UT_PR2 5015.13 BOOL  ; FRA NODE1
V4255_INN 2532.10 BOOL
V4255_INN_PR 5124.14 BOOL  ; TIL NODE1
V4255_UT 2232.10 BOOL
V4255_UT_N5 2847.13 BOOL
V4255_UT_PR2 5015.14 BOOL  ; FRA NODE1
V4305_INN 2552.06 BOOL
V4305_UT 2252.06 BOOL
V4305_UT_N5 2800.07 BOOL  ; Z
V4401_INN 2551.11 BOOL
V4401_UT 2251.11 BOOL
V4402_INN 2551.12 BOOL
V4402_UT 2251.12 BOOL
V4501_INN 2551.13 BOOL  ; V4520_BAK
V4501_UT 2251.13 BOOL  ; V4520_BAK
V4502_INN 2551.14 BOOL
V4502_UT 2251.14 BOOL
V4503_INN 2551.15 BOOL
V4503_UT 2251.15 BOOL
V4504_INN 2552.00 BOOL
V4504_UT 2252.00 BOOL  ; V2702.08
V4505_INN 2552.01 BOOL
V4505_UT 2252.01 BOOL
V4511_INN 2552.05 BOOL
V4511_UT 2252.05 BOOL
V4520_INN 2552.02 BOOL
V4520_UT 2252.02 BOOL
V4550_INN 2552.03 BOOL
V4550_UT 2252.03 BOOL
V4551_INN 2552.04 BOOL
V4551_UT 2252.04 BOOL
V510_NEDRE 2224.07 BOOL
V510_OEVRE 2224.06 BOOL
V520_NEDRE 2224.09 BOOL
V520_OEVRE 2224.08 BOOL
V5280_INN 2539.15 BOOL
V5280_UT 2239.15 BOOL
V5281_INN 2540.00 BOOL
V5281_UT 2240.00 BOOL
V530_NEDRE 2224.11 BOOL
V530_OEVRE 2224.10 BOOL
V540_NEDRE 2224.13 BOOL
V540_OEVRE 2224.12 BOOL
V7047_UT 2903.09 BOOL  ; FRA NODE1    LUTDOSERING T98  VST90-UHT
V7056_UT 2903.10 BOOL  ; FRA NODE1    DOSERING DESINFEKSJON T97  VST90-UHT
V8001_INN 2502.00 BOOL  ; VANNDREN_K2
V8001_UT 2202.00 BOOL  ; VANNDREN_VST80-K1
V8001_UT_PR2_07 5009.00 BOOL  ; TIL PROFIBUS
V8002_INN 2502.02 BOOL  ; VANNDREN_K2
V8002_INN_DR2_07 5116.01 BOOL  ; FRA PROFIBUS
V8002_UT 2202.02 BOOL  ; VANNDREN_K2
V8002_UT_PR2_07 5009.01 BOOL  ; TIL PROFIBUS
V8003_HJ 932.01 BOOL
V8003_INN 2502.04 BOOL  ; VANNDREN_K3
V8003_INN_DR2_07 5116.02 BOOL  ; FRA PROFIBUS
V8003_UT 2202.04 BOOL  ; VANNDREN_K3
V8003_UT_PR2_07 5009.02 BOOL  ; TIL PROFIBUS
V8007_UT 2209.09 BOOL  ; Z
V8008_UT_N 2209.10 BOOL  ; Z
V8011_UT 2202.01 BOOL  ; L
V8011_UT_PR2 5009.12 BOOL  ; TIL PROFIBUS
V8014_D_MEM D25013 CHANNEL
V8014_HJ1 952.00 BOOL
V8014_I_MEM D25012 CHANNEL
V8014_MANUELL 1000.03 BOOL
V8014_PRS D8700 UINT  ; SKAL_RETTES_TIL_K2_KOND_ERVERDI
V8014_PRS_MID D9700 CHANNEL
V8014_P_MEM D25011 CHANNEL
V8014_UT_AN D1406 CHANNEL  ; Z
V8018_INN 2518.05 BOOL
V8018_UT 2218.05 BOOL
V8019_UT 2205.04 BOOL  ; VST80-K1-RETUR TIL GRM.
V8021_UT 2202.03 BOOL  ; VST80-K1-TUR LUFTVENTIL
V8021_UT_PR2 5009.13 BOOL  ; TIL PROFIBUS
V8022_INN 2507.10 BOOL  ; Z
V8022_UT 2207.10 BOOL  ; Z
V8023_INN 2507.12 BOOL  ; Z
V8023_UT 2207.12 BOOL  ; Z
V8024_D_MEM D25033 CHANNEL
V8024_HJ1 952.01 BOOL
V8024_INN 2507.13 BOOL  ; Z
V8024_I_MEM D25032 CHANNEL
V8024_MANUELL 1000.04 BOOL
V8024_PRS D8702 CHANNEL
V8024_PRS_MID D9702 CHANNEL
V8024_P_MEM D25031 CHANNEL
V8024_UT 2207.13 BOOL  ; Z
V8024_UT_AN D1408 CHANNEL  ; Z
V8025_INN 2507.14 BOOL  ; Z
V8025_UT 2207.14 BOOL  ; Z
V8026_INN 2508.01 BOOL  ; Z
V8026_UT 2208.01 BOOL  ; Z
V8028_INN 2518.06 BOOL
V8028_UT 2218.06 BOOL
V8031_UT 2202.05 BOOL  ; VST80-K1-TUR LUFTVENTIL
V8031_UT_PR2 5009.14 BOOL  ; TIL PROFIBUS
V8034_AUTOPAADRAG D4268 CHANNEL
V8034_D_MEM D25053 CHANNEL
V8034_HJ1 952.02 BOOL
V8034_I_MEM D25052 CHANNEL
V8034_MANUELL 1000.05 BOOL
V8034_PRS D8704 CHANNEL  ; XXXVST80_K2_B8022_ER_TT
V8034_PRSR D8832 CHANNEL
V8034_PRS_REG_6 D4266 CHANNEL
V8034_P_MEM D25051 CHANNEL
V8034_UT_AN D1410 CHANNEL  ; Z
V8036_AUTO 1053.10 BOOL
V8036_HJ1 903.00 BOOL
V8036_MAN 1003.10 BOOL
V8036_UT 2202.06 BOOL  ; Z
V8037_AUTO 1053.11 BOOL
V8037_HJ1 913.00 BOOL
V8037_MAN 1003.11 BOOL
V8037_UT 2202.07 BOOL  ; Z
V8038_INN 2518.07 BOOL
V8038_UT 2218.07 BOOL
V8041_INN 2508.10 BOOL  ; Z
V8041_UT 2208.10 BOOL  ; Z
V8043_AUTO 1053.12 BOOL
V8043_HJ1 923.00 BOOL
V8043_INN 2521.07 BOOL  ; Z
V8043_MAN 1003.12 BOOL
V8043_UT 2202.08 BOOL  ; Z
V8043_UT_N 2221.07 BOOL  ; Z
V8045_INN 2507.15 BOOL  ; Z
V8045_UT 2207.15 BOOL  ; Z
V8046_INN 2517.15 BOOL  ; Z
V8046_UT 2217.15 BOOL  ; Z
V8047_INN 2510.00 BOOL  ; Z
V8047_UT 2210.00 BOOL  ; Z
V8048_INN 2510.01 BOOL  ; Z
V8048_UT_N 2210.01 BOOL  ; Z
V8050_INN 2508.11 BOOL  ; Z
V8050_UT 2208.11 BOOL  ; Z
V8051_INN 2508.12 BOOL  ; Z
V8051_UT 2208.12 BOOL  ; Z
V8053_INN 2510.04 BOOL  ; Z
V8053_UT 2210.04 BOOL  ; Z
V8053_V8054_VEKSL 1318.10 BOOL
V8054_INN 2510.05 BOOL  ; Z
V8054_UT_N 2210.05 BOOL  ; Z
V8060_INN 2503.00 BOOL  ; Z
V8060_UT 2203.00 BOOL  ; Z
V8061_INN 2503.06 BOOL  ; Z
V8061_UT 2203.06 BOOL  ; Z
V8062_INN 2503.03 BOOL  ; Z
V8062_UT 2203.03 BOOL  ; Z
V8063_INN 2503.09 BOOL  ; Z
V8063_UT 2203.09 BOOL  ; Z
V8064_INN 2503.12 BOOL  ; Z
V8064_UT 2203.12 BOOL  ; Z
V8065_INN 2504.02 BOOL  ; Z
V8065_UT 2204.02 BOOL  ; Z
V8066_INN 2503.15 BOOL  ; Z
V8066_UT 2203.15 BOOL  ; Z
V8067_INN 2504.05 BOOL  ; Z
V8067_UT 2204.05 BOOL  ; Z
V8070_INN 2503.01 BOOL  ; Z
V8070_UT 2203.01 BOOL  ; Z
V8071_INN 2503.07 BOOL  ; Z
V8071_UT 2203.07 BOOL  ; Z
V8072_INN 2503.04 BOOL  ; Z
V8072_UT 2203.04 BOOL  ; Z
V8073_INN 2503.10 BOOL  ; Z
V8073_UT 2203.10 BOOL  ; Z
V8074_INN 2503.13 BOOL  ; Z
V8074_UT 2203.13 BOOL  ; Z
V8075_INN 2504.03 BOOL  ; Z
V8075_UT 2204.03 BOOL  ; Z
V8076_INN 2504.00 BOOL  ; Z
V8076_UT 2204.00 BOOL  ; Z
V8077_INN 2504.06 BOOL  ; Z
V8077_UT 2204.06 BOOL  ; Z
V80_K1_V_VEKSL_B_H 1306.11 BOOL  ; VEKSLING AV TURVENTILER I VASK BIL OGHENGER
V80_K2_V_VEKSL_B_H 1316.11 BOOL  ; VEKSLING AV TURVENTILER I VASK BIL OGHENGER
V80_K3_V_VEKSL_B_H 1326.11 BOOL  ; VEKSLING AV TURVENTILER I VASK BIL OGHENGER
V8101_INN 2500.00 BOOL  ; Z
V8101_INN_PR2 5127.00 BOOL  ; TIL NODE1
V8101_UT 2200.00 BOOL  ; Z
V8101_UT_PR2 5018.00 BOOL  ; FRA NODE1
V8102_INN 2500.01 BOOL  ; Z
V8102_INN_PR2 5127.01 BOOL  ; TIL NODE1
V8102_UT 2200.01 BOOL  ; Z
V8102_UT_PR2 5018.01 BOOL  ; FRA NODE1
V8103_INN 2500.02 BOOL  ; Z
V8103_INN_PR2 5127.02 BOOL  ; TIL NODE1
V8103_UT 2200.02 BOOL  ; Z
V8103_UT_PR2 5018.02 BOOL  ; FRA NODE1
V8111_HJ1 931.05 BOOL
V8111_HJ2 931.06 BOOL
V8111_INN 2501.00 BOOL  ; Z
V8111_INN_PR2 5127.03 BOOL  ; TIL NODE1
V8111_UT 2201.00 BOOL
V8111_UT_PR2 5018.03 BOOL  ; FRA NODE1
V8112_HJ1 941.05 BOOL
V8112_HJ2 941.06 BOOL
V8112_INN 2501.01 BOOL  ; Z
V8112_INN_PR2 5127.04 BOOL  ; TIL NODE1
V8112_UT 2201.01 BOOL  ; Z
V8112_UT_PR2 5018.04 BOOL  ; FRA NODE1
V8113_HJ1 951.05 BOOL
V8113_HJ2 951.06 BOOL
V8113_INN 2501.02 BOOL  ; Z
V8113_INN_PR2 5127.05 BOOL  ; TIL NODE1
V8113_UT 2201.02 BOOL  ; Z
V8113_UT_PR2 5018.05 BOOL  ; FRA NODE1
V8120_INN 2517.09 BOOL  ; Z
V8120_TON T0400 BOOL  ; FORSINER  STENGING AV SLUK FRA PASTEURER
V8120_UT 2217.09 BOOL  ; Z
V8121_AUTO 1052.13 BOOL
V8121_UT 2201.12 BOOL  ; Z
V8121_UT_PR2_07 5009.09 BOOL  ; TIL PROFIBUS
V8201_HJ 903.02 BOOL
V8201_INN 2500.03 BOOL  ; Z
V8201_INN_PR2 5127.06 BOOL  ; TIL NODE1
V8201_UT 2200.03 BOOL
V8201_UT_PR2 5018.06 BOOL  ; FRA NODE1
V8202_HJ 913.02 BOOL
V8202_INN 2500.04 BOOL  ; Z
V8202_INN_PR2 5127.07 BOOL  ; TIL NODE1
V8202_UT 2200.04 BOOL  ; Z
V8202_UT_PR2 5018.07 BOOL  ; FRA NODE1
V8203_HJ 923.02 BOOL
V8203_INN 2500.05 BOOL  ; Z
V8203_INN_PR2 5127.08 BOOL  ; TIL NODE1
V8203_UT 2200.05 BOOL  ; Z
V8203_UT_PR2 5018.08 BOOL  ; FRA NODE1
V8204_INN 2517.12 BOOL  ; Z
V8204_INN_PR2 5127.09 BOOL  ; TIL NODE1
V8204_UT 2217.12 BOOL  ; Z
V8204_UT_PR2 5018.09 BOOL  ; FRA NODE1
V8211_FORS_INN T0153 BOOL  ; TID SOM FORSINKER  VENTIL AAPNING TIL T82 NAAR LUTKONSENTASJON ER OK FOERSTE GANG
V8211_HJ1 931.07 BOOL
V8211_HJ2 931.08 BOOL
V8211_INN 2501.03 BOOL  ; Z
V8211_INN_PR2 5127.10 BOOL  ; TIL NODE1
V8211_UT 2201.03 BOOL
V8211_UT_PR2 5018.10 BOOL  ; FRA NODE1
V8212_FORS_INN T0155 BOOL  ; TID SOM FORSINKER  VENTIL AAPNING TIL T82 NAAR LUTKONSENTASJON ER OK FOERSTE GANG
V8212_HJ1 931.10 BOOL
V8212_HJ2 931.11 BOOL
V8212_INN 2501.04 BOOL  ; Z
V8212_INN_PR2 5127.11 BOOL  ; TIL NODE1
V8212_UT 2201.04 BOOL  ; Z
V8212_UT_PR2 5018.11 BOOL  ; FRA NODE1
V8213_FORS_INN T0156 BOOL  ; TID SOM FORSINKER  VENTIL AAPNING TIL T82 NAAR LUTKONSENTASJON ER OK FOERSTE GANG
V8213_HJ1 941.10 BOOL
V8213_HJ2 941.11 BOOL
V8213_INN 2501.05 BOOL  ; Z
V8213_INN_PR2 5127.12 BOOL  ; TIL NODE1
V8213_UT 2201.05 BOOL  ; Z
V8213_UT_PR2 5018.12 BOOL  ; FRA NODE1
V8214_INN 2517.10 BOOL  ; Z
V8214_INN_PR2 5127.13 BOOL  ; TIL NODE1
V8214_UT 2217.10 BOOL  ; Z
V8214_UTFORSINK T0443 BOOL  ; FORSINKER  VENTILSTENGNING
V8214_UT_PR2 5018.13 BOOL  ; FRA NODE1
V8221_AUTO 1052.14 BOOL
V8221_UT 2201.13 BOOL  ; Z
V8221_UT_PR2_07 5009.03 BOOL  ; TIL PROFIBUS
V8222_UT_N 2209.05 BOOL  ; Z
V8222_UT_PR2_07 5009.10 BOOL  ; TIL PROFIBUS
V8223_AUTO 1052.00 BOOL
V8223_UT 2200.13 BOOL  ; Z
V8223_UT_PR2_07 5009.08 BOOL  ; TIL PROFIBUS
V8224_AVTID T0061 BOOL
V8224_AVTID_T 0061 NUMBER
V8224_UT 2226.00 BOOL
V8301_INN_PR2 5127.14 BOOL  ; TIL NODE1
V8301_UT_PR2 5018.14 BOOL  ; FRA NODE1
V8302_INN_PR2 5127.15 BOOL  ; TIL NODE1
V8302_UT_PR2 5018.15 BOOL  ; FRA NODE1
V8304_INN 2517.13 BOOL
V8304_INN_PR2 5128.01 BOOL  ; TIL NODE1
V8304_UT 2217.13 BOOL  ; Z
V8304_UT_PR2 5019.01 BOOL  ; FRA NODE1
V8314_INN 2517.11 BOOL  ; Z
V8314_INN_PR2 5128.05 BOOL  ; TIL NODE1
V8314_UT 2217.11 BOOL  ; Z
V8314_UTFORSINK T0444 BOOL  ; FORSINKER  VENTILSTENGNING
V8314_UT_PR2 5019.05 BOOL  ; FRA NODE1
V8321_AUTO 1052.15 BOOL
V8321_UT 2201.14 BOOL  ; Z
V8321_UT_PR2_07 5009.04 BOOL  ; TIL PROFIBUS
V8322_UT_N 2209.06 BOOL  ; Z
V8322_UT_PR2_07 5009.11 BOOL  ; TIL PROFIBUS
V8323_AUTO 1052.01 BOOL
V8323_UT 2200.14 BOOL  ; Z
V8323_UT_PR2_07 5009.07 BOOL  ; TIL PROFIBUS
V8324_AVTID T0062 BOOL
V8324_UT 2226.01 BOOL
V8401_HJ1 903.03 BOOL
V8401_HJ2 903.04 BOOL
V8401_INN 2500.06 BOOL  ; Z
V8401_INN_PR2 5128.06 BOOL  ; TIL NODE1
V8401_UT 2200.06 BOOL
V8401_UT_PR2 5019.06 BOOL  ; FRA NODE1
V8402_HJ1 913.03 BOOL
V8402_HJ2 913.04 BOOL
V8402_INN 2500.07 BOOL  ; Z
V8402_INN_PR2 5128.07 BOOL  ; TIL NODE1
V8402_UT 2200.07 BOOL  ; Z
V8402_UT_PR2 5019.07 BOOL  ; FRA NODE1
V8403_HJ1 923.03 BOOL
V8403_HJ2 923.04 BOOL
V8403_INN 2500.08 BOOL  ; Z
V8403_INN_PR2 5128.08 BOOL  ; TIL NODE1
V8403_UT 2200.08 BOOL  ; Z
V8403_UT_PR2 5019.08 BOOL  ; FRA NODE1
V8411_HJ1 931.09 BOOL
V8411_INN 2501.06 BOOL  ; Z
V8411_INN_PR2 5128.09 BOOL  ; TIL NODE1
V8411_UT 2201.06 BOOL
V8411_UT_PR2 5019.09 BOOL  ; FRA NODE1
V8412_HJ1 931.12 BOOL
V8412_INN 2501.07 BOOL  ; Z
V8412_INN_PR2 5128.10 BOOL  ; TIL NODE1
V8412_UT 2201.07 BOOL  ; Z
V8412_UT_PR2 5019.10 BOOL  ; FRA NODE1
V8413_HJ1 941.12 BOOL
V8413_INN 2501.08 BOOL  ; Z
V8413_INN_PR2 5128.11 BOOL  ; TIL NODE1
V8413_UT 2201.08 BOOL  ; Z
V8413_UT_PR2 5019.11 BOOL  ; FRA NODE1
V8421_AUTO 1053.00 BOOL
V8421_UT 2201.10 BOOL
V8421_UT_PR2_07 5009.06 BOOL  ; TIL PROFIBUS
V8422_INN 2515.01 BOOL  ; Z
V8422_UT_N 2215.01 BOOL  ; Z
V8422_UT_PR2_07 5009.05 BOOL  ; TIL PROFIBUS
V8423_INN 2515.02 BOOL  ; Z
V8423_UT_N 2215.02 BOOL  ; Z
V8424_UT 2226.02 BOOL
V9010_UT_N5 2859.00 BOOL
V9011_UT_N5 2859.01 BOOL
V9012_UT_N5 2859.02 BOOL
V9018_INN 2518.08 BOOL
V9018_UT 2218.08 BOOL
V9021_INN 2507.04 BOOL  ; Z
V9021_UT 2207.04 BOOL  ; Z
V9022_INN 2507.07 BOOL  ; Z
V9022_UT 2207.07 BOOL  ; Z
V9023_INN 2507.08 BOOL  ; Z
V9023_UT 2207.08 BOOL  ; Z
V9024_INN 2507.11 BOOL  ; Z
V9024_UT 2207.11 BOOL  ; Z
V9025_INN 2507.09 BOOL  ; Z
V9025_UT 2207.09 BOOL  ; Z
V9028_INN 2518.09 BOOL
V9028_UT 2218.09 BOOL
V9038_INN 2518.10 BOOL
V9038_UT 2218.10 BOOL
V9060_INN 2506.00 BOOL  ; Z
V9060_UT 2206.00 BOOL  ; Z
V9061_INN 2506.06 BOOL  ; Z
V9061_UT 2206.06 BOOL  ; Z
V9062_INN 2506.03 BOOL  ; Z
V9062_UT 2206.03 BOOL  ; Z
V9063_INN 2506.09 BOOL  ; Z
V9063_UT 2206.09 BOOL  ; Z
V9064_INN 2506.12 BOOL  ; Z
V9064_UT 2206.12 BOOL  ; Z
V9065_INN 2507.02 BOOL  ; Z
V9065_UT 2207.02 BOOL  ; Z
V9066_INN 2506.15 BOOL  ; Z
V9066_UT 2206.15 BOOL  ; Z
V9067_INN 2507.05 BOOL  ; Z
V9067_UT 2207.05 BOOL  ; Z
V9070_INN 2506.01 BOOL  ; Z
V9070_UT 2206.01 BOOL  ; Z
V9071_INN 2506.07 BOOL  ; Z
V9071_UT 2206.07 BOOL  ; Z
V9072_INN 2506.04 BOOL  ; Z
V9072_UT 2206.04 BOOL  ; Z
V9073_INN 2506.10 BOOL  ; Z
V9073_UT 2206.10 BOOL  ; Z
V9074_INN 2506.13 BOOL  ; Z
V9074_UT 2206.13 BOOL  ; Z
V9075_INN 2507.03 BOOL  ; Z
V9075_UT 2207.03 BOOL  ; Z
V9076_INN 2507.00 BOOL  ; Z
V9076_UT 2207.00 BOOL  ; Z
V9077_INN 2507.06 BOOL  ; Z
V9077_UT 2207.06 BOOL  ; Z
VACUUM_P4001_1_INN 2603.12 BOOL
VACUUM_P4001_2_INN 2603.13 BOOL
VANND_L11_V0303 720.00 BOOL
VANND_L11_V0312 720.03 BOOL
VANND_L11_V0403 720.01 BOOL
VANND_L11_V0503 720.02 BOOL
VANND_L12_V0303 720.08 BOOL
VANND_L12_V0322 720.11 BOOL
VANND_L12_V0403 720.09 BOOL
VANND_L12_V0503 720.10 BOOL
VANND_L21_V0305 722.00 BOOL
VANND_L21_V0332 722.03 BOOL
VANND_L21_V0405 722.01 BOOL
VANND_L21_V0505 722.02 BOOL
VANND_L22_V0305 722.08 BOOL
